MC_GearIn_1(
	Master:= Axis_Spindle  , 
	Slave:=AXIS_1   , 
	Execute:=R_TRIG_5.Q OR ((R_TRIG_1.Q OR R_TRIG_2.Q OR R_TRIG_3.Q) AND HandWheel_3Y) , 
	RatioNumerator:=iMolecule , 
	RatioDenominator:= iDenominator, 
	Acceleration:= 500, 
	Deceleration:= 800, 
	Jerk:= , 
	//BufferMode:= , 
	InGear=> %MX500.5, 
	Busy=> , 
	//Active=> , 
	CommandAborted=> , 
	Error=> , 
	ErrorID=> );
//2轴启动啮合
MC_GearIn_2(
	Master:= Axis_Spindle, 
	Slave:=AXIS_2 , 
	Execute:=R_TRIG_6.Q OR ((R_TRIG_1.Q OR R_TRIG_2.Q OR R_TRIG_3.Q) AND HandWheel_4X) , 
	RatioNumerator:=iMolecule , 
	RatioDenominator:= iDenominator, 
	Acceleration:= 500, 
	Deceleration:= 800, 
	Jerk:= , 
	//BufferMode:= , 
	InGear=> , 
	Busy=> , 
	//Active=> , 
	CommandAborted=> , 
	Error=> , 
	ErrorID=> );
//3轴启动啮合
MC_GearIn_3(
	Master:= Axis_Spindle, 
	Slave:=AXIS_3 , 
	Execute:= R_TRIG_7.Q OR ((R_TRIG_1.Q OR R_TRIG_2.Q OR R_TRIG_3.Q) AND HandWheel_5Z), 
	RatioNumerator:=iMolecule , 
	RatioDenominator:= iDenominator, 
	Acceleration:= 500, 
	Deceleration:= 800, 
	Jerk:= , 
	//BufferMode:= , 
	InGear=> , 
	Busy=> , 
	//Active=> , 
	CommandAborted=> , 
	Error=> , 
	ErrorID=> );
//4轴启动啮合
MC_GearIn_4(
	Master:= Axis_Spindle, 
	Slave:=AXIS_4 , 
	Execute:=  R_TRIG_8.Q OR ((R_TRIG_1.Q OR R_TRIG_2.Q OR R_TRIG_3.Q) AND HandWheel_6X), 
	RatioNumerator:=iMolecule , 
	RatioDenominator:= iDenominator, 
	Acceleration:= 500, 
	Deceleration:= 800, 
	Jerk:= , 
	//BufferMode:= , 
	InGear=> , 
	Busy=> , 
	//Active=> , 
	CommandAborted=> , 
	Error=> , 
	ErrorID=> );
//5轴启动啮合
MC_GearIn_5(
	Master:= Axis_Spindle, 
	Slave:=AXIS_5 , 
	Execute:= R_TRIG_9.Q OR ((R_TRIG_1.Q OR R_TRIG_2.Q OR R_TRIG_3.Q) AND HandWheel_7Y), 
	RatioNumerator:=iMolecule , 
	RatioDenominator:= iDenominator, 
	Acceleration:= 500, 
	Deceleration:= 800, 
	Jerk:= , 
	//BufferMode:= , 
	InGear=> , 
	Busy=> , 
	//Active=> , 
	CommandAborted=> , 
	Error=> , 
	ErrorID=> );
//6轴启动啮合
MC_GearIn_6(
	Master:= Axis_Spindle, 
	Slave:=AXIS_6 , 
	Execute:= R_TRIG_10.Q OR ((R_TRIG_1.Q OR R_TRIG_2.Q OR R_TRIG_3.Q) AND HandWheel_8Y), 
	RatioNumerator:=iMolecule , 
	RatioDenominator:= iDenominator, 
	Acceleration:= 500, 
	Deceleration:= 800, 
	Jerk:= , 
	//BufferMode:= , 
	InGear=> , 
	Busy=> , 
	//Active=> , 
	CommandAborted=> , 
	Error=> , 
	ErrorID=> );
//7轴启动啮合
MC_GearIn_7(
	Master:= Axis_Spindle, 
	Slave:=AXIS_7 , 
	Execute:= R_TRIG_11.Q OR ((R_TRIG_1.Q OR R_TRIG_2.Q OR R_TRIG_3.Q) AND HandWheel_9X), 
	RatioNumerator:=iMolecule , 
	RatioDenominator:= iDenominator, 
	Acceleration:= 500, 
	Deceleration:= 800, 
	Jerk:= , 
	//BufferMode:= , 
	InGear=> , 
	Busy=> , 
	//Active=> , 
	CommandAborted=> , 
	Error=> , 
	ErrorID=> );
//8轴启动啮合
MC_GearIn_8(
	Master:= Axis_Spindle, 
	Slave:=AXIS_8 , 
	Execute:= R_TRIG_12.Q OR ((R_TRIG_1.Q OR R_TRIG_2.Q OR R_TRIG_3.Q) AND HandWheel_10Z), 
	RatioNumerator:=iMolecule , 
	RatioDenominator:= iDenominator, 
	Acceleration:= 500, 
	Deceleration:= 800, 
	Jerk:= , 
	//BufferMode:= , 
	InGear=> , 
	Busy=> , 
	//Active=> , 
	CommandAborted=> , 
	Error=> , 
	ErrorID=> );
//9轴启动啮合
MC_GearIn_9(
	Master:= Axis_Spindle, 
	Slave:=AXIS_9 , 
	Execute:=  R_TRIG_13.Q OR ((R_TRIG_1.Q OR R_TRIG_2.Q OR R_TRIG_3.Q) AND HandWheel_11Y), 
	RatioNumerator:=iMolecule , 
	RatioDenominator:= iDenominator, 
	Acceleration:= 500, 
	Deceleration:= 800, 
	Jerk:= , 
	//BufferMode:= , 
	InGear=> , 
	Busy=> , 
	//Active=> , 
	CommandAborted=> , 
	Error=> , 
	ErrorID=> );

Error :=MC_GearIn_1.Error OR MC_GearIn_2.Error OR MC_GearIn_3.Error OR MC_GearIn_4.Error OR MC_GearIn_5.Error OR MC_GearIn_6.Error OR MC_GearIn_7.Error OR MC_GearIn_8.Error OR MC_GearIn_9.Error ;  
ErrorID :=MC_GearIn_1.ErrorID OR MC_GearIn_2.ErrorID OR MC_GearIn_3.ErrorID OR MC_GearIn_4.ErrorID OR MC_GearIn_5.ErrorID OR MC_GearIn_6.ErrorID OR MC_GearIn_7.ErrorID OR MC_GearIn_8.ErrorID OR MC_GearIn_9.ErrorID ;  

//1轴断开齿合
MC_GearOut_1(Slave:=AXIS_1 , Execute:= F_TRIG_1.Q AND MC_GearIn_1.InGear , Done=> xStop_1 , Busy=> , Error=> , ErrorID=> );

//2轴断开齿合
MC_GearOut_2(Slave:=AXIS_2 , Execute:= F_TRIG_2.Q AND MC_GearIn_2.InGear , Done=> xStop_2 , Busy=> , Error=> , ErrorID=> );

//3轴断开齿合
MC_GearOut_3(Slave:=AXIS_3 , Execute:= F_TRIG_3.Q AND MC_GearIn_3.InGear , Done=> xStop_3 , Busy=> , Error=> , ErrorID=> );


//4轴断开齿合
MC_GearOut_4(Slave:=AXIS_4 , Execute:= F_TRIG_4.Q AND MC_GearIn_4.InGear , Done=> xStop_4 , Busy=> , Error=> , ErrorID=> );


//5轴断开齿合
MC_GearOut_5(Slave:=AXIS_5 , Execute:= F_TRIG_5.Q AND MC_GearIn_5.InGear , Done=> xStop_5 , Busy=> , Error=> , ErrorID=> );


//6轴断开齿合
MC_GearOut_6(Slave:=AXIS_6 , Execute:= F_TRIG_6.Q AND MC_GearIn_6.InGear , Done=> xStop_6 , Busy=> , Error=> , ErrorID=> );


//7轴断开齿合
MC_GearOut_7(Slave:=AXIS_7 , Execute:= F_TRIG_7.Q AND MC_GearIn_7.InGear , Done=> xStop_7 , Busy=> , Error=> , ErrorID=> );


//8断开齿合
MC_GearOut_8(Slave:=AXIS_8 , Execute:= F_TRIG_8.Q AND MC_GearIn_8.InGear , Done=> xStop_8 , Busy=> , Error=> , ErrorID=> );


//9轴断开齿合
MC_GearOut_9(Slave:=AXIS_9 , Execute:= F_TRIG_9.Q AND MC_GearIn_9.InGear , Done=> xStop_9 , Busy=> , Error=> , ErrorID=> );

END_FUNCTION_BLOCK

// Device/Application/30_Ethercat任务/PLC_CNC
PROGRAM PLC_CNC
VAR
	SMC_Interpolator: SMC_Interpolator;
	SMC_ControlAxisByPos1: SMC_ControlAxisByPos;
	SMC_ControlAxisByPos2: SMC_ControlAxisByPos;
	SMC_ControlAxisByPos3: SMC_ControlAxisByPos;
	SMC_TRAFO_Gantry3: SMC_TRAFO_Gantry3;
	SMC_TRAFOF_Gantry3: SMC_TRAFOF_Gantry3;
	SMC_NCDecoder_0: SMC_NCDecoder;
	SMC_CheckVelocities: SMC_CheckVelocities;
	SMC_SmoothPath: SMC_SmoothPath;
	SR: SR;
	RS: RS;
END_VAR
VAR // added by the converter: edge detectors and wires of the graphical bodies
    _w1, _w2, _w3 : BOOL;
    _w4, _w5 : ANY;
END_VAR

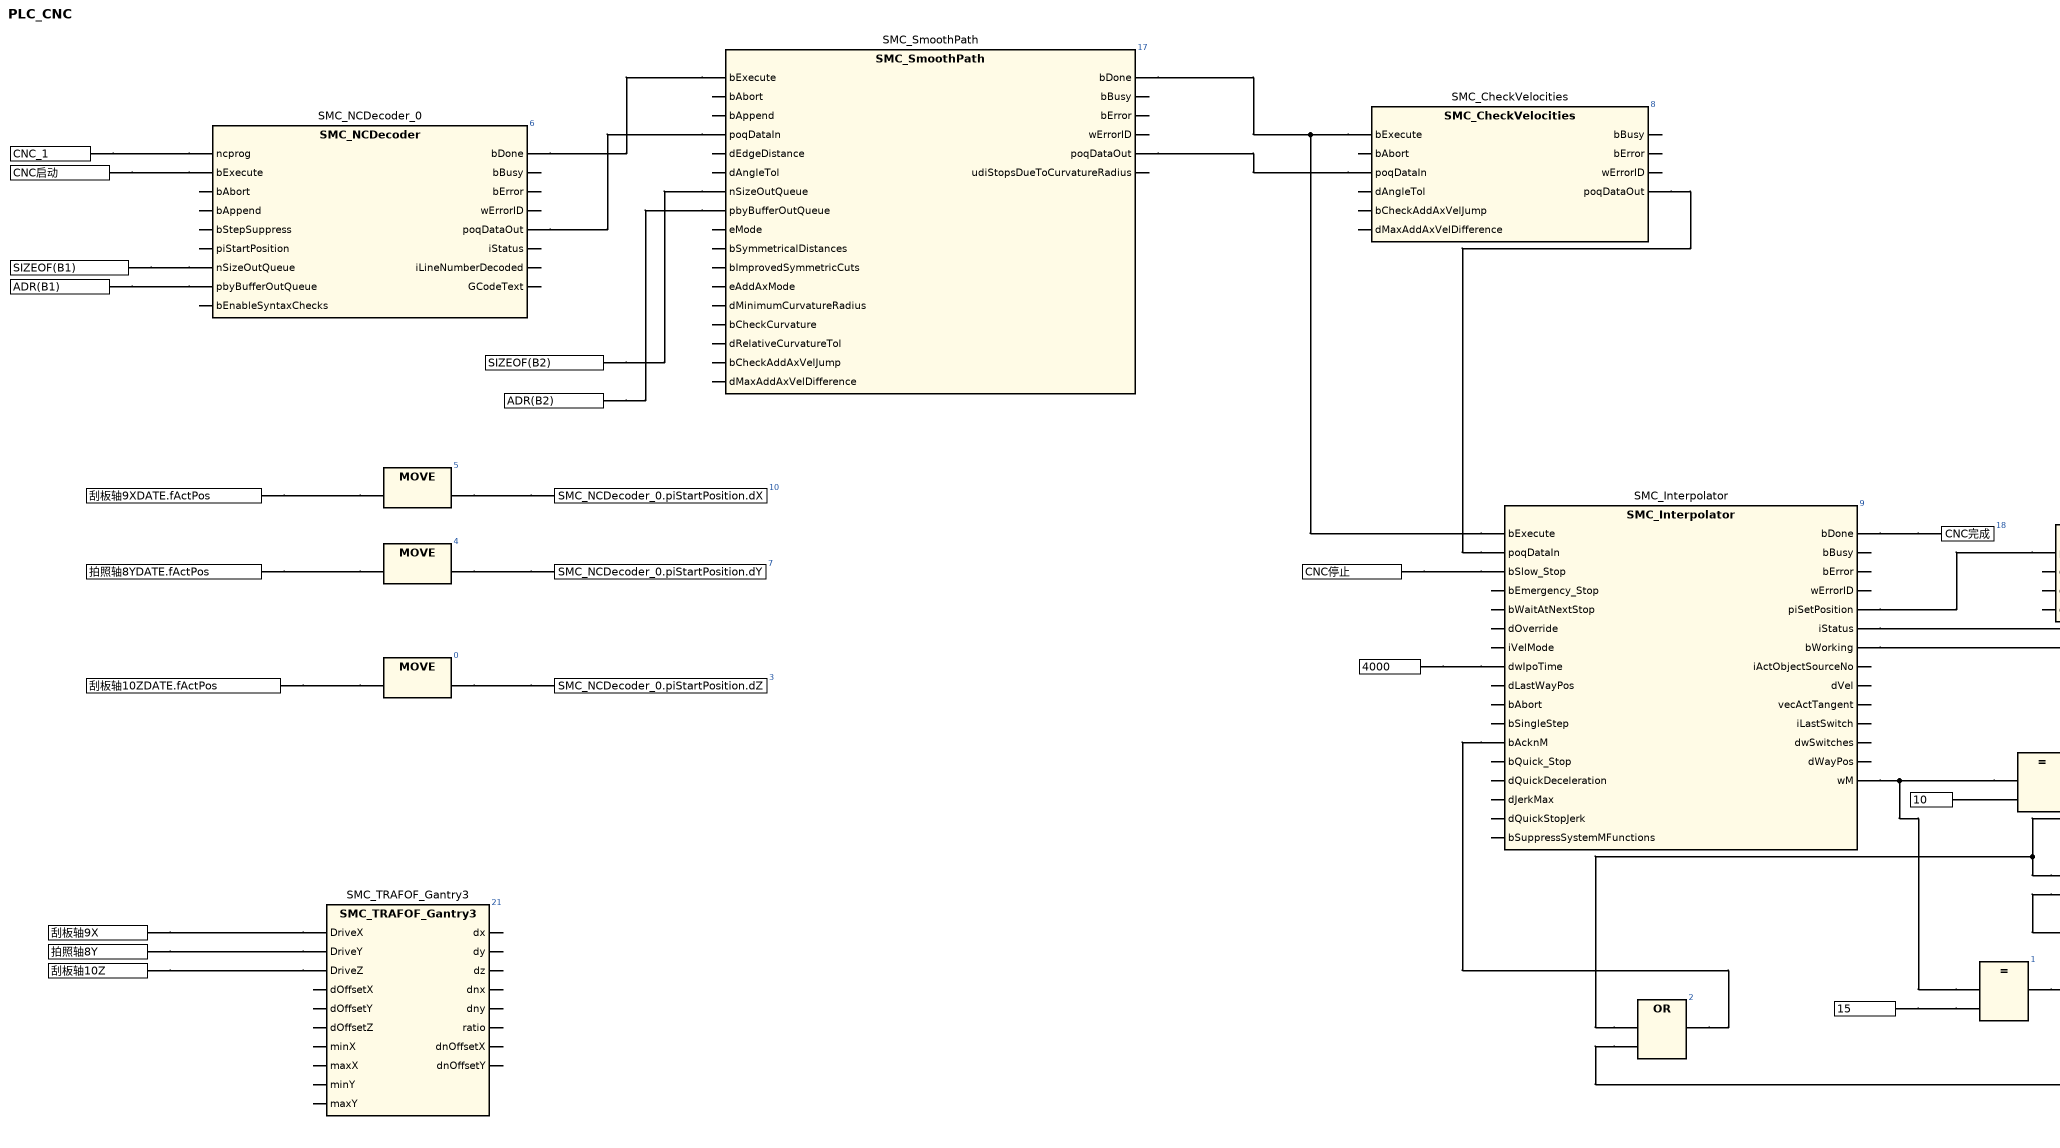
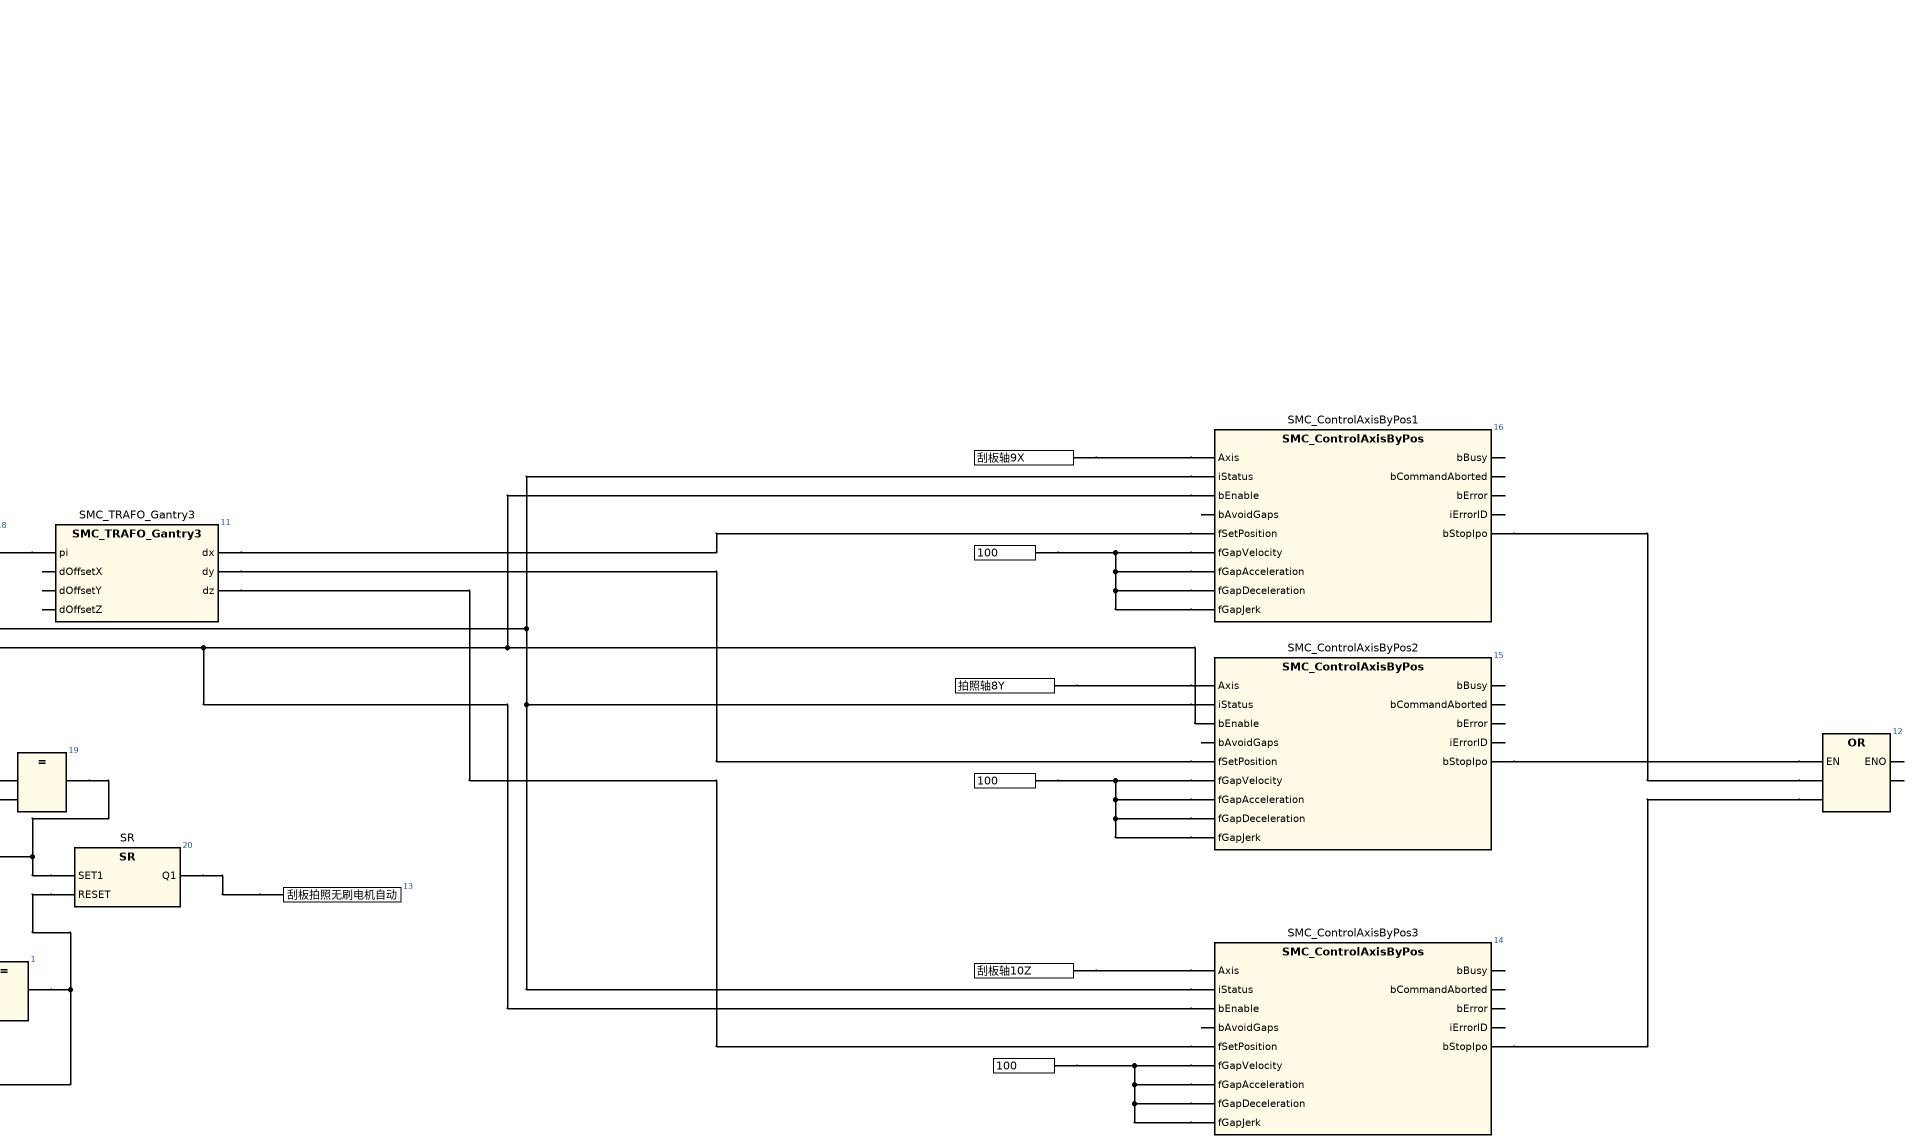
// note: 4 stored wires end on pins the file does not list and are not shown
_w1 := SMC_Interpolator.wM = 15;
_w3 := _w2 OR _w1;
SMC_NCDecoder_0.piStartPosition.dZ := 刮板轴10ZDATE.fActPos;
_w4 := 拍照轴8YDATE.fActPos;
_w5 := 刮板轴9XDATE.fActPos;
SMC_NCDecoder_0(
    ncprog := CNC_1,
    bExecute := CNC启动,
    nSizeOutQueue := SIZEOF(B1),
    pbyBufferOutQueue := ADR(B1)); // SMC_NCDecoder
SMC_NCDecoder_0.piStartPosition.dY := _w4;
SMC_CheckVelocities(bExecute := SMC_SmoothPath.bDone, poqDataIn := SMC_SmoothPath.poqDataOut);
SMC_Interpolator(
    bExecute := SMC_SmoothPath.bDone,
    poqDataIn := SMC_CheckVelocities.poqDataOut,
    bSlow_Stop := CNC停止,
    dwIpoTime := 4000,
    bAcknM := _w3);
SMC_NCDecoder_0.piStartPosition.dX := _w5;
SMC_TRAFO_Gantry3(pi := SMC_Interpolator.piSetPosition);
IF SMC_ControlAxisByPos2.bStopIpo THEN (* SMC_ControlAxisByPos1.bStopIpo OR SMC_ControlAxisByPos3.bStopIpo; result not used *) END_IF
刮板拍照无刷电机自动 := SR.Q1;
SMC_ControlAxisByPos3(
    Axis := 刮板轴10Z,
    iStatus := SMC_Interpolator.iStatus,
    bEnable := SMC_Interpolator.bWorking,
    fSetPosition := SMC_TRAFO_Gantry3.dz,
    fGapVelocity := 100,
    fGapAcceleration := 100,
    fGapDeceleration := 100,
    fGapJerk := 100); // SMC_ControlAxisByPos
SMC_ControlAxisByPos2(
    Axis := 拍照轴8Y,
    iStatus := SMC_Interpolator.iStatus,
    bEnable := SMC_Interpolator.bWorking,
    fSetPosition := SMC_TRAFO_Gantry3.dy,
    fGapVelocity := 100,
    fGapAcceleration := 100,
    fGapDeceleration := 100,
    fGapJerk := 100); // SMC_ControlAxisByPos
SMC_ControlAxisByPos1(
    Axis := 刮板轴9X,
    iStatus := SMC_Interpolator.iStatus,
    bEnable := SMC_Interpolator.bWorking,
    fSetPosition := SMC_TRAFO_Gantry3.dx,
    fGapVelocity := 100,
    fGapAcceleration := 100,
    fGapDeceleration := 100,
    fGapJerk := 100); // SMC_ControlAxisByPos
SMC_SmoothPath(
    bExecute := SMC_NCDecoder_0.bDone,
    poqDataIn := SMC_NCDecoder_0.poqDataOut,
    nSizeOutQueue := SIZEOF(B2),
    pbyBufferOutQueue := ADR(B2));
CNC完成 := SMC_Interpolator.bDone;
_w2 := SMC_Interpolator.wM = 10;
SR(SET1 := _w2, RESET := _w1);
SMC_TRAFOF_Gantry3(DriveX := 刮板轴9X, DriveY := 拍照轴8Y, DriveZ := 刮板轴10Z);

END_PROGRAM

// Device/Application/40_Man/PLC_MainPRG
PROGRAM PLC_MainPRG

VAR
	PLC_Mode_0: FB_Mode;
	TON_1: TON;
	RB_Control_0: FB_RB_Control;
	TON_0: TON;
	TON_2: TON;
	TON_3: TON;
	SysHC_ModbusTcpSlaveDiagnose_0: SysHC_ModbusTcpSlaveDiagnose;
	点样step: INT;
	打样伺服移动step: INT;
END_VAR

IF 点样测试 THEN
	CASE 打样伺服移动step OF
		
		0:
			点样轴6XDATE.fAbsTarget:=HMI_点样轴6X.position[2];        //起始位
			点样轴6XDATE.xMoveAbs:=TRUE;
			打样伺服移动step:=20;
		20:
			IF 点样轴6XDATE.bAbMoveDone THEN
				
				打样伺服移动step:=30;
				点样轴6XDATE.xMoveAbs:=FALSE;
			END_IF
		30:
			点样轴6XDATE.fAbsTarget:=HMI_点样轴6X.position[3];             //终点位
			点样轴6XDATE.xMoveAbs:=TRUE;
			打样伺服移动step:=40;
		40:
			IF 点样轴6XDATE.bAbMoveDone THEN
				
				打样伺服移动step:=0;
				点样轴6XDATE.xMoveAbs:=FALSE;
			END_IF
			
	END_CASE
ELSE
	打样伺服移动step:=0;
END_IF







A00_设备状态显示及控制 ();

A20_机器人();
%MW1000:=0;

PLC_Cyinder_气缸动作();

CASE MODE_State OF
	EN_功能块状态.运行:
		A10_上下料伺服流程 ();
		Sample_point_sampling_上样点样();
		Collection_process_收集流程();
		Expand_process_展开流程();
		Photo_scraper_拍照刮板();
		Robotic_Process_机器人流程();
		Develop_TankDrain();
	IF NOT 上料进料传感器 THEN
		Alarm.2:=TRUE;
	END_IF
	IF NOT 下料出料传感器 THEN
		Alarm.3:=TRUE;
	END_IF
END_CASE




//所有状态复位
TON_3(IN:=复位,PT:=T#5S );
IF NOT 急停 OR TON_3.Q THEN
	A30_急停();
END_IF





//升降伺服流程
IF MODE_State<>1 THEN
	伺服上料_Setp:=0;
	伺服下料_Setp:=0;
END_IF






//检测MODBUS通讯
SysHC_ModbusTcpSlaveDiagnose_0(
	xEnable:=TRUE , 
	strSlaveIP:= '192.168.0.15', 
	xValid=> , 
	xBusy=> , 
	xError=> , 
	eErrorID=> , 
	stDiagData=>ModbusTcpError );

ACTION A30_急停:

伺服上料_Setp:=0;
伺服下料_Setp:=0;
//收集工位
收集下压气缸手动:=FALSE;
收集下压气缸自动:=FALSE;
收集夹持气缸手动:=FALSE;
收集夹持气缸自动:=FALSE;
收集升降气缸手动:=FALSE;
收集升降气缸自动:=FALSE;
收集伸缩气缸手动:=FALSE;
收集伸缩气缸自动:=FALSE;
收集进液手动:=FALSE;
收集进液自动:=FALSE;
收集排液手动:=FALSE;
收集排液自动:=FALSE;
收集正压排液手动:=FALSE;
收集正压排液自动:=FALSE;
溶液收集瓶定位手动:=FALSE;
收集工位允许放收集瓶:=FALSE;
收集工位允许放收集器:=FALSE;
收集工位允许机器人退出工位:=FALSE;
收集工位允许机器人取收集瓶放暂存工位:=FALSE;
收集工位允许取收集器:=FALSE;
收集工位机器人取收集器放回暂存工位:=FALSE;
collect_prepare_OK:=FALSE;
collect_OK:=FALSE;
收集工位放收集器完成:=FALSE;
收集工位放收集瓶完成:=FALSE;
收集工位放收集器到工位:=FALSE;

收集工位机器人退出完成:=FALSE;

收集工位机器人放收集瓶到暂存工位完成:=FALSE;

收集工位机器人到达收集器位置:=FALSE;
//展开工位
expand_initialization_OK:=FALSE;
Expand_Group_clean_OK:=FALSE;
Expand_up_liquid_OK:=FALSE;
Expand_silica_gel_plate_OK:=FALSE;
展开工位允许放硅胶板:=FALSE;
展开工位允许取硅胶板:=FALSE;
展开工位机器人到达准备点:=FALSE;
展开工位机器人放硅胶板完成:=FALSE;
展开工位取硅胶板完成:=FALSE;
展开工位允许放硅胶板1:=FALSE;
展缸1气缸1手动:=FALSE;
展缸1气缸1自动:=FALSE;
展缸1进液电池阀1手动:=FALSE;
展缸1进液电池阀1自动:=FALSE;
展缸1排液电池阀1手动:=FALSE;
展缸1排液电池阀1自动:=FALSE;
展缸1吹气电池阀1手动:=FALSE;
展缸1吹气电池阀1自动:=FALSE;
展缸1气缸2手动:=FALSE;
展缸1气缸2自动:=FALSE;
展缸1进液电池阀2手动:=FALSE;
展缸1进液电池阀2自动:=FALSE;
展缸1排液电池阀2手动:=FALSE;
展缸1排液电池阀2自动:=FALSE;
展缸1吹气电池阀2手动:=FALSE;
展缸1吹气电池阀2自动:=FALSE;
展缸1气缸3手动:=FALSE;
展缸1气缸3自动:=FALSE;
展缸1进液电池阀3手动:=FALSE;
展缸1进液电池阀3自动:=FALSE;	
展缸1排液电池阀3手动:=FALSE;
展缸1排液电池阀3自动:=FALSE;
展缸1吹气电池阀3手动:=FALSE;
展缸1吹气电池阀3自动:=FALSE;
展缸1气缸4手动:=FALSE;
展缸1气缸4自动:=FALSE;
展缸1进液电池阀4手动:=FALSE;
展缸1进液电池阀4自动:=FALSE;	
展缸1排液电池阀4手动:=FALSE;
展缸1排液电池阀4自动:=FALSE;
展缸1吹气电池阀4手动:=FALSE;
展缸1吹气电池阀4自动:=FALSE;
展缸2气缸1手动:=FALSE;
展缸2气缸1自动:=FALSE;
展缸2进液电池阀1手动:=FALSE;
展缸2进液电池阀1自动:=FALSE;
展缸2排液电池阀1手动:=FALSE;
展缸2排液电池阀1自动:=FALSE;
展缸2吹气电池阀1手动:=FALSE;
展缸2吹气电池阀1自动:=FALSE;
展缸2气缸2手动:=FALSE;
展缸2气缸2自动:=FALSE;
展缸2进液电池阀2手动:=FALSE;
展缸2进液电池阀2自动:=FALSE;
展缸2排液电池阀2手动:=FALSE;
展缸2排液电池阀2自动:=FALSE;
展缸2吹气电池阀2手动:=FALSE;
展缸2吹气电池阀2自动:=FALSE;
展缸2气缸3手动:=FALSE;
展缸2气缸3自动:=FALSE;
展缸2进液电池阀3手动:=FALSE;
展缸2进液电池阀3自动:=FALSE;	
展缸2排液电池阀3手动:=FALSE;
展缸2排液电池阀3自动:=FALSE;
展缸2吹气电池阀3手动:=FALSE;
展缸2吹气电池阀3自动:=FALSE;
展缸2气缸4手动:=FALSE;
展缸2气缸4自动:=FALSE;
展缸2进液电池阀4手动:=FALSE;
展缸2进液电池阀4自动:=FALSE;	
展缸2排液电池阀4手动:=FALSE;
展缸2排液电池阀4自动:=FALSE;
展缸2吹气电池阀4手动:=FALSE;
展缸2吹气电池阀4自动:=FALSE;
Expand_Step:=0;
//拍照刮板
刮板拍照真空自动:=FALSE;
刮板拍照真空手动:=FALSE;
刮板拍照无刷电机手动:=FALSE;
刮板拍照无刷电机自动:=FALSE;
刮板拍照定位气缸手动:=FALSE;
刮板拍照定位气缸自动:=FALSE;
粉末收集器定位手动:=FALSE;
粉末收集器定位自动:=FALSE;
刮板拍照遮光气缸手动:=FALSE;
刮板拍照遮光气缸自动:=FALSE;
刮板拍照旋转气缸手动:=FALSE;
刮板拍照旋转气缸自动:=FALSE;
刮板拍照下压气缸手动:=FALSE;
刮板拍照下压气缸自动:=FALSE;
拍照工位允许放硅胶板:=FALSE;
拍照工位允许放收集器:=FALSE;
拍照工位机器人退出工位:=FALSE;
拍照工位允许取收集器:=FALSE;
拍照工位机器人退出:=FALSE;
拍照工位放硅胶板完成 := FALSE;
 scrape_IsLast := FALSE;       // ★ 新增		
拍照工位机器人到达夹持位 := FALSE;
scrape_PhotoMode:=0;
拍照工位机器人退出工位完成 := FALSE;
刮板拍照工位站位符:=FALSE;
拍照工位机器人到达收集器夹持位 := FALSE;
scrape_Step:=0;
拍照工位机器人退出完成 := FALSE;
拍照工位允许取硅胶板放废料区 := FALSE;
拍照工位允许取硅胶板去展开 := FALSE;
拍照工位机器人取硅胶板完成 := FALSE;
scrape_WaitConfirm := FALSE;
Camera_scraper_initialization_OK:=FALSE;
Photo_preparation_completed_OK:=FALSE;
Scraper_collection_completed:=FALSE;
Robot_completes_material_retrieval:=FALSE;	
取拍照硅胶完step:=0;

//上样点样
上样定位手动:=FALSE;
上样定位自动:=FALSE;
上样点样三通电池阀手动:=FALSE;
上样点样三通电池阀自动:=FALSE;
上样吹气手动:=FALSE;
上样吹气自动:=FALSE;
打样瓶上料轴3YDATE.fAbsTarget:=0;
点样轴6XDATE.fAbsTarget:=0;
点样轴7YDATE.fAbsTarget:=0;
上样轴4X轴DATE.fAbsTarget:=0;
上样轴5Z轴DATE.fAbsTarget:=0;
上样点样允许放硅胶板:=FALSE;
点样轴7YDATE.xMoveAbs:=FALSE;
点样轴6XDATE.xMoveAbs:=FALSE;
上样轴5Z轴DATE.xMoveAbs:=FALSE;
上样轴4X轴DATE.xMoveAbs:=FALSE;
打样瓶上料轴3YDATE.xMoveAbs:=FALSE;
Sampling_Spray_sample_OK:=FALSE;
Sampling_liquid_absorption:=FALSE;
Sampling_preparation_OK:=FALSE;
上样点样允许取硅胶板:=FALSE;
上样点样放硅胶板完成:=FALSE;
大真空泵站位[11]:=FALSE;
大真空泵自动:=FALSE;
Sampling_Step:=0;

//机器人
Execute:=0;
FunctionID:=0;
ParameterList1:=0;
ParameterList2:=0;
ParameterList3:=0;
ParameterList4:=0;
ParameterList5:=0;
ParameterList6:=0;
ParameterList7:=0;
ParameterList8:=0;
ParameterList9:=0;
ParameterList10:=0;

RO_ParameterList1:=0;
RO_ParameterList2:=0;
RO_ParameterList4:=0;
RO_ParameterList5:=0;
RO_ParameterList6:=0;
RO_ParameterList7:=0;
RO_ParameterList8:=0;
RO_ParameterList9:=0;
RO_ParameterList10:=0;
升降上料机器人取料完成:=FALSE;
泵站位符:=FALSE;
上样料架报警:=FALSE;
取工具setp:=0;
取工具完成:=FALSE;
取升降硅胶板step:=0;
取升降硅胶板完成:=FALSE;
放点样硅胶板step:=0;
放点样硅胶板完成:=FALSE;
取点样硅胶板step:=0;
取点样硅胶板完成:=FALSE;
放展缸硅胶板完成:=FALSE;
放展缸硅胶板step:=0;
取展缸硅胶板step:=0;
取展缸硅胶板完成:=FALSE;
放拍照硅胶板完成:=FALSE;
放拍照硅胶板step:=0;
取收集器组放暂存工位step:=0;
取收集瓶组放暂存工位完成:=FALSE;
取暂存收集器放刮板位完成:=FALSE;
取暂存收集器放刮板位step:=0;
取刮板收集器放到收集工位完成:=FALSE;
取刮板收集器放到收集工位step:=0;
取暂存收集瓶放收集工位step:=0;
取暂存收集瓶放收集工位完成:=FALSE;
取收集器放暂存工位完成:=FALSE;
取收集器放暂存工位step:=0;
取刮板硅胶板放废料区step:=0;
取刮板硅胶板放废料区完成:=FALSE;
取暂存收集器组放仓库完成:=FALSE;
取暂存收集器组放仓库step:=0;
取收集器组放暂存工位完成:=FALSE;
取收集瓶组放暂存工位step:=0;
取暂存收集瓶组放仓库完成:=FALSE;
取暂存收集瓶组放仓库step:=0;
取收集瓶放暂存工位step:=0;
取收集瓶放暂存工位完成:=FALSE;
机器人流程:=0;
溶液收集瓶定位自动:=FALSE;
溶液收集瓶定位手动:=FALSE;
END_ACTION

ACTION A20_机器人:
//机器人远程控制
RB_Control_0(
    PowerOn := RB_使能状态, 
    PowerOnOut =>RB_上使能 , 

    ResetOut =>RB_复位 , 

    Reset := 复位, 

    StartCmd := 启动, 
    StopCmd :=  TON_3.Q OR NOT 急停, 
    PauseCmd := NOT 停止, 
    RobotRunning := RB_运行中, 
    RobotStopped :=RB_停止中 , 
    RobotPaused :=RB_暂停中 , 
    RobotAlarm :=RB_报警中 , 
    StartOut =>RB_启动 , 
    StopOut => RB_停止, 
    PauseOut =>  RB_暂停, 
    StatusRun => , 
    StatusStop => , 
    StatusPause => , 
    StatusAlarm => , 

	);
END_ACTION

ACTION A00_设备状态显示及控制:
//PLC模式切换
PLC_Mode_0(
    bWarning_alarm := cyinderAlarm<>0 OR Alarm<>0 OR 上样料架报警 OR ModbusTcpError.byDiagData>0, 

	xStart:= 启动 OR PLCStart, 
	xStop:=NOT  停止 OR PLCStop, 
	xReset:=复位  , 
	xAutoMode:=手自动  , 
	xFault:=伺服报警 OR ECAT掉站报警 OR 伺服未回原点报警, 
	xEmergency:= 急停 , 
	bRed=>三色灯红  , 
	bYellow=> 三色灯黄, 
	bGreen=> 三色灯绿, 
	bBuzzer=> 蜂鸣器 , 
	iState=>MODE_STATE  , 
	bAuto=>ManualAuto  );
	
	//伺服报错
IF   玻璃上料轴1ZDATE.bError OR 玻璃上料轴2ZDATE.bError OR 打样瓶上料轴3YDATE.bError OR 点样轴6XDATE.bError OR 点样轴7YDATE.bError OR 拍照轴8YDATE.bError OR 刮板轴9XDATE.bError OR 刮板轴10ZDATE.bError OR 地轨轴11YDATE.bError OR 上样轴4X轴DATE.bError OR 上样轴5Z轴DATE.bError THEN
	伺服报警:=TRUE;
END_IF
   //伺服报错复位
IF 复位 THEN
	伺服报警:=FALSE;
	伺服未回原点报警:=FALSE;
	Alarm:=0;
	cyinderAlarm:=0;
	上样料架报警:=FALSE;
END_IF


IF NOT 玻璃上料轴1ZDATE.bHomed OR NOT 玻璃上料轴2ZDATE.bHomed OR NOT 打样瓶上料轴3YDATE.bHomed OR NOT 点样轴6XDATE.bHomed OR NOT 点样轴7YDATE.bHomed OR NOT 拍照轴8YDATE.bHomed OR NOT 刮板轴9XDATE.bHomed OR NOT 刮板轴10ZDATE.bHomed  OR NOT 地轨轴11YDATE.bHomed OR NOT 上样轴4X轴DATE.bHomed OR NOT 上样轴5Z轴DATE.bHomed THEN
	伺服未回原点报警:=TRUE ;
END_IF
END_ACTION

ACTION A10_上下料伺服流程:
//初始化
IF MODE_State =4 OR  初始化  THEN

		玻璃上料轴1ZDATE.fAbsTarget :=0;
		玻璃上料轴1ZDATE.xMoveAbs:=TRUE;
		玻璃上料轴1ZDATE.xJogPos :=FALSE;
		升降上料伺服允许取料 :=FALSE ;
		升降上料伺服下降完成 :=FALSE ;
		伺服上料_Setp:=0;
		伺服上料_Setp:=0;
		升降下料伺服允许放料  :=FALSE ;
		玻璃上料轴2ZDATE.xJogNeg :=FALSE;
		玻璃上料轴2ZDATE.xJogPos :=FALSE;
		升降上料机器人取料完成:=FALSE;
END_IF



//上料流程
IF MODE_State =1 THEN     //自动模式下
	IF 玻璃上料轴1ZDATE.bHomed AND 玻璃升降接近开关1 AND 上料进料传感器 AND 伺服上料_Setp=0 AND NOT Alarm.0 AND 升降上料完成 THEN
		伺服上料_Setp :=1;
	END_IF
	
    CASE 伺服上料_Setp OF
    	1 :
			IF NOT 玻璃升降光电开关1 AND 玻璃上料轴1ZDATE.fActPos<514  THEN
				Z1JOG_pos :=TRUE;
				ELSE
				Z1JOG_pos :=FALSE;
				伺服上料_Setp:=10;
			END_IF
   
	   10:
		   IF 玻璃升降光电开关1 THEN
		   	升降上料伺服允许取料 :=TRUE;
			伺服上料_Setp:=20;
		   END_IF
		   
	   20:
		   IF 升降上料机器人已吸住物料 THEN
		   	玻璃上料轴1ZDATE.fRelTarget :=-5.0;
			玻璃上料轴1ZDATE.xMoveRel :=TRUE;
			升降上料机器人已吸住物料:=FALSE;
			伺服上料_Setp:=30;
		   END_IF
	   30:
		   IF 玻璃上料轴1ZDATE .bReMoveDone  THEN
		   	升降上料伺服下降完成 :=TRUE ;
			玻璃上料轴1ZDATE.xMoveRel :=FALSE;
			伺服上料_Setp:=40;
		   END_IF
	   40:
		   IF 升降上料机器人取料完成  THEN
		   	升降上料伺服下降完成 :=FALSE ;
			升降上料伺服允许取料 :=FALSE ;
			升降上料机器人取料完成:=FALSE;
			伺服上料_Setp:=1;
		   END_IF 
    END_CASE
	
	IF 玻璃上料轴1ZDATE.fActPos>=510.0 AND  玻璃升降光电开关1 AND  NOT 玻璃升降接近开关1 THEN
		Alarm.0:=TRUE;                                             //上料机构无物料
		升降上料完成:=FALSE;
		玻璃上料轴1ZDATE.fAbsTarget :=0;
		玻璃上料轴1ZDATE.xMoveAbs:=TRUE;
		Z1JOG_pos :=FALSE;
		升降上料伺服允许取料 :=FALSE ;
		升降上料伺服下降完成 :=FALSE ;
		伺服上料_Setp:=0;
	END_IF
	IF 玻璃上料轴1ZDATE .bAbMoveDone  THEN
		玻璃上料轴1ZDATE.xMoveAbs:=FALSE;
		升降上料机器人放料完成:=FALSE;
    END_IF
	
	
END_IF
//下料流程
IF MODE_State =1 THEN     //自动模式下
	IF 玻璃上料轴2ZDATE.bHomed  AND 下料出料传感器 AND 伺服下料_Setp=0 AND NOT Alarm.1 AND 升降下料完成 THEN
		伺服下料_Setp :=1;
	END_IF
	
    CASE 伺服下料_Setp  OF
    	1 :
			IF NOT 玻璃升降光电开关2 AND 玻璃上料轴2ZDATE.fActPos<510  THEN
				Z2JOG_POS :=TRUE;
				
				ELSE
				Z2JOG_POS :=FALSE;
				伺服下料_Setp:=10;
			END_IF
   
	   10:
		   IF 玻璃升降光电开关2 THEN
			   Z2JOG_NEG :=TRUE;
			   伺服下料_Setp:=15;
		   END_IF
	   15:
		   IF NOT 玻璃升降光电开关2  THEN
				升降下料伺服允许放料  :=TRUE;
				Z2JOG_NEG :=FALSE;
				伺服下料_Setp:=20;
		   END_IF
			  
	   
	   20:
		   IF 升降下料机器人放废料完成 AND 玻璃升降光电开关2 AND 玻璃升降接近开关2 THEN
		   	Z2JOG_NEG :=TRUE;
			升降下料伺服允许放料  :=FALSE ;
			升降下料机器人放废料完成:=FALSE;
			伺服下料_Setp:=30;
		   END_IF
		  
	   30:
		   IF NOT 玻璃升降光电开关2 THEN
		   	Z2JOG_NEG :=FALSE;
			取刮板硅胶板放废料区完成:=FALSE;
			伺服下料_Setp:=15;
		   END_IF
	  
    END_CASE
	
	IF 玻璃上料轴2ZDATE.fActPos<=0 AND 玻璃升降光电开关1 THEN
		Alarm.1:=TRUE;                                           //下料机构已满料
		升降下料完成:=FALSE;
		伺服下料_Setp:=0;
		升降下料伺服允许放料  :=FALSE ;
		Z2JOG_NEG :=FALSE;
		Z2JOG_POS :=FALSE;
		玻璃上料轴2ZDATE.fAbsTarget :=0;
		玻璃上料轴2ZDATE.xMoveAbs:=TRUE;
		伺服下料_Setp:=0;
	END_IF
	IF 玻璃上料轴2ZDATE .bAbMoveDone  THEN
		玻璃上料轴2ZDATE.xMoveAbs:=FALSE;
		升降下料伺服允许放料  :=FALSE ;
    END_IF
END_IF
END_ACTION

END_PROGRAM

// Device/Application/40_Man/PLC_Cyinder_气缸动作
PROGRAM PLC_Cyinder_气缸动作
VAR
	cylinder_0: FB_cylinder;
	cylinder_1: FB_cylinder;
	cylinder_2: FB_cylinder;
	cylinder_3 :FB_cylinder ;
	cylinder_4 :FB_cylinder ;
	cylinder_5 :FB_cylinder ;
	cylinder_6 :FB_cylinder ;
	cylinder_7 :FB_cylinder ;
	cylinder_8 :FB_cylinder ;
	cylinder_9 :FB_cylinder ;
	cylinder_10 :FB_cylinder ;
	cylinder_11 :FB_cylinder ;
	cylinder_12 :FB_cylinder ;
	cylinder_13 :FB_cylinder ;
	cylinder_14 :FB_cylinder ;
	cylinder_15 :FB_cylinder ;
	cylinder_16 :FB_cylinder ;
	cylinder_17 :FB_cylinder ;
	cylinder_18 :FB_cylinder ;
	cylinder_19 :FB_cylinder ;
	cylinder_20 :FB_cylinder ;
	cylinder_21 :FB_cylinder ;
	cylinder_22 :FB_cylinder ;
	cylinder_23 :FB_cylinder ;
	cylinder_24 :FB_cylinder ;
	cylinder_25 :FB_cylinder ;
	cylinder_26 :FB_cylinder ;
	cylinder_27 :FB_cylinder ;
	cylinder_28 :FB_cylinder ;
	cylinder_29 :FB_cylinder ;
	cylinder_30 :FB_cylinder ;
	cylinder_31 :FB_cylinder ;
	cylinder_32 :FB_cylinder ;
	cylinder_33 :FB_cylinder ;
	cylinder_34 :FB_cylinder ;
	cylinder_35 :FB_cylinder ;
	cylinder_36 :FB_cylinder ;
	cylinder_37 :FB_cylinder ;
	cylinder_38 :FB_cylinder ;
	cylinder_39 :FB_cylinder ;
	cylinder_40 :FB_cylinder ;
	cylinder_41 :FB_cylinder ;
	cylinder_42 :FB_cylinder ;
	cylinder_43 :FB_cylinder ;
	cylinder_44 :FB_cylinder ;
	cylinder_45 :FB_cylinder ;
	cylinder_46 :FB_cylinder ;
	cylinder_47 :FB_cylinder ;
	cylinder_48 :FB_cylinder ;
	cylinder_49 :FB_cylinder ;
	cylinder_50 :FB_cylinder ;
END_VAR

//气缸动作
//展缸1气缸1
cylinder_0(
    xManualRetract := , 
    xAutoRetract := , 
    yValve2 => , 
    cylinder_type := 0, 

	xManualAuto:=ManualAuto  , 
	xManualExtend:=展缸1气缸1手动 , 
	xAutoExtend:= 展缸1气缸1自动, 
	xReset:=复位  , 
	xPosExtend:= 展缸1气缸1原点, 
	xPosRetract:= 展缸1气缸1动点 , 
	tTimeout:= T#5S, 
	yValve1=> 展缸1气缸1 , 
	bAlarm=> cyinderAlarm.0);
//展缸1气缸2
cylinder_1(
    xManualRetract := , 
    xAutoRetract := , 
    yValve2 => , 
    cylinder_type :=0 , 

	xManualAuto:=ManualAuto  , 
	xManualExtend:=展缸1气缸2手动 , 
	xAutoExtend:= 展缸1气缸2自动, 
	xReset:=复位  , 
	xPosExtend:= 展缸1气缸2原点, 
	xPosRetract:= 展缸1气缸2动点 , 
	tTimeout:= T#5S, 
	yValve1=> 展缸1气缸2, 
	bAlarm=> cyinderAlarm.1);
//展缸1气缸3
cylinder_2(
    xManualRetract := , 
    xAutoRetract := , 
    yValve2 => , 
    cylinder_type := 0, 

	xManualAuto:=ManualAuto  , 
	xManualExtend:=展缸1气缸3手动 , 
	xAutoExtend:= 展缸1气缸3自动, 
	xReset:=复位  , 
	xPosExtend:= 展缸1气缸3原点, 
	xPosRetract:= 展缸1气缸3动点 , 
	tTimeout:= T#5S, 
	yValve1=> 展缸1气缸3, 
	bAlarm=> cyinderAlarm.2);
//展缸1气缸4
cylinder_3(
    xManualRetract := , 
    xAutoRetract := , 
    yValve2 => , 
    cylinder_type :=0 , 

	xManualAuto:=ManualAuto  , 
	xManualExtend:=展缸1气缸4手动 , 
	xAutoExtend:= 展缸1气缸4自动, 
	xReset:=复位  , 
	xPosExtend:= 展缸1气缸4原点, 
	xPosRetract:= 展缸1气缸4动点 , 
	tTimeout:= T#5S, 
	yValve1=> 展缸1气缸4, 
	bAlarm=> cyinderAlarm.3);
//展缸2气缸1
cylinder_4(
    xManualRetract := , 
    xAutoRetract := , 
    yValve2 => , 
    cylinder_type := 0, 

	xManualAuto:=ManualAuto  , 
	xManualExtend:=展缸2气缸1手动 , 
	xAutoExtend:= 展缸2气缸1自动, 
	xReset:=复位  , 
	xPosExtend:= 展缸2气缸1原点, 
	xPosRetract:= 展缸2气缸1动点 , 
	tTimeout:= T#5S, 
	yValve1=> 展缸2气缸1, 
	bAlarm=> cyinderAlarm.4);
//展缸2气缸2
cylinder_5(
    xManualRetract := , 
    xAutoRetract := , 
    yValve2 => , 
    cylinder_type :=0 , 

	xManualAuto:=ManualAuto  , 
	xManualExtend:=展缸2气缸2手动 , 
	xAutoExtend:= 展缸2气缸2自动, 
	xReset:=复位  , 
	xPosExtend:= 展缸2气缸2原点, 
	xPosRetract:= 展缸2气缸2动点 , 
	tTimeout:= T#5S, 
	yValve1=> 展缸2气缸2, 
	bAlarm=> cyinderAlarm.5);
//展缸2气缸3
cylinder_6(
    xManualRetract := , 
    xAutoRetract := , 
    yValve2 => , 
    cylinder_type := 0, 

	xManualAuto:=ManualAuto  , 
	xManualExtend:=展缸2气缸3手动 , 
	xAutoExtend:= 展缸2气缸3自动, 
	xReset:=复位  , 
	xPosExtend:= 展缸2气缸3原点, 
	xPosRetract:= 展缸2气缸3动点 , 
	tTimeout:= T#5S, 
	yValve1=> 展缸2气缸3, 
	bAlarm=> cyinderAlarm.6);
//展缸2气缸4
cylinder_7(
    xManualRetract := , 
    xAutoRetract := , 
    yValve2 => , 
    cylinder_type := 0, 

	xManualAuto:=ManualAuto  , 
	xManualExtend:=展缸2气缸4手动 , 
	xAutoExtend:= 展缸2气缸4自动, 
	xReset:=复位  , 
	xPosExtend:= 展缸2气缸4原点, 
	xPosRetract:= 展缸2气缸4动点 , 
	tTimeout:= T#5S, 
	yValve1=> 展缸2气缸4, 
	bAlarm=> cyinderAlarm.7);
//大真空泵
cylinder_8(
    xManualRetract := , 
    xAutoRetract := , 
    yValve2 => , 
    cylinder_type :=0 , 

	xManualAuto:=ManualAuto  , 
	xManualExtend:= 大真空泵手动, 
	xAutoExtend:= 大真空泵自动, 
	xReset:=复位  , 
	xPosExtend:= , 
	xPosRetract:=  , 
	tTimeout:= , 
	yValve1=> 大真空泵, 
	bAlarm=> );
//收集平台下压气缸
cylinder_9(
    xManualRetract := , 
    xAutoRetract := , 
    yValve2 => , 
    cylinder_type := 0, 

	xManualAuto:=ManualAuto  , 
	xManualExtend:= 收集下压气缸手动, 
	xAutoExtend:= 收集下压气缸自动, 
	xReset:=复位  , 
	xPosExtend:=收集平台下压气缸原点 , 
	xPosRetract:= 收集下压气缸手动 OR 收集下压气缸自动, 
	tTimeout:= T#5S, 
	yValve1=> 收集下压气缸 , 
	bAlarm=> cyinderAlarm.8);
//收集平台夹持气缸
cylinder_10(
    xManualRetract := , 
    xAutoRetract := , 
    yValve2 => , 
    cylinder_type := 0, 

	xManualAuto:=ManualAuto  , 
	xManualExtend:= 收集夹持气缸手动, 
	xAutoExtend:= 收集夹持气缸自动, 
	xReset:=复位  , 
	xPosExtend:=收集平台夹持气缸原点 , 
	xPosRetract:= 收集平台夹持气缸动点, 
	tTimeout:= T#5S, 
	yValve1=> 收集夹持气缸  , 
	bAlarm=> cyinderAlarm.9);	
//收集平台升降气缸
cylinder_11(
    xManualRetract := , 
    xAutoRetract := , 
    yValve2 => , 
    cylinder_type := 0, 

	xManualAuto:=ManualAuto  , 
	xManualExtend:= 收集升降气缸手动, 
	xAutoExtend:= 收集升降气缸自动, 
	xReset:=复位  , 
	xPosExtend:=收集平台升降气缸原点 , 
	xPosRetract:= 收集平台升降气缸动点, 
	tTimeout:= T#5S, 
	yValve1=> 收集升降气缸   , 
	bAlarm=> cyinderAlarm.10);	
//收集平台伸缩气缸
cylinder_12(
    xManualRetract := , 
    xAutoRetract := , 
    yValve2 => , 
    cylinder_type :=0 , 

	xManualAuto:=ManualAuto  , 
	xManualExtend:= 收集伸缩气缸手动, 
	xAutoExtend:= 收集伸缩气缸自动, 
	xReset:=复位, 
	xPosExtend:=收集平台推出气缸原点, 
	xPosRetract:= 收集平台推出气缸动点, 
	tTimeout:= T#5S, 
	yValve1=> 收集伸缩气缸, 
	bAlarm=> cyinderAlarm.11);		
//刮板拍照遮光气缸
cylinder_13(
    xManualRetract := , 
    xAutoRetract := , 
    yValve2 => , 
    cylinder_type :=0 , 

	xManualAuto:=ManualAuto  , 
	xManualExtend:= 刮板拍照遮光气缸手动, 
	xAutoExtend:=刮板拍照遮光气缸自动 , 
	xReset:=复位  , 
	xPosExtend:=刮板拍照遮光气缸上位 , 
	xPosRetract:= 刮板拍照遮光气缸下位, 
	tTimeout:= T#5S, 
	yValve1=>  刮板拍照遮光气缸, 
	bAlarm=> cyinderAlarm.12);		
//刮板拍照旋转气缸
cylinder_14(
    xManualRetract := , 
    xAutoRetract := , 
    yValve2 => , 
    cylinder_type := 0, 

	xManualAuto:=ManualAuto  , 
	xManualExtend:= 刮板拍照旋转气缸手动 AND 刮板轴9XDATE.fActPos>330, 
	xAutoExtend:=刮板拍照旋转气缸自动 , 
	xReset:=复位  , 
	xPosExtend:=刮板拍照旋转气缸原点  , 
	xPosRetract:= 刮板拍照旋转气缸动点, 
	tTimeout:= T#5S, 
	yValve1=>  刮板拍照旋转气缸   , 
	bAlarm=> cyinderAlarm.13);		
//刮板拍照下压气缸
cylinder_15(
    xManualRetract := , 
    xAutoRetract := , 
    yValve2 => , 
    cylinder_type := 0, 

	xManualAuto:=ManualAuto  , 
	xManualExtend:= 刮板拍照下压气缸手动, 
	xAutoExtend:=刮板拍照下压气缸自动 , 
	xReset:=复位  , 
	xPosExtend:=刮板拍照下压气缸上位, 
	xPosRetract:=刮板拍照下压气缸手动 OR 刮板拍照下压气缸自动 , 
	tTimeout:= T#5S, 
	yValve1=>  刮板拍照下压气缸, 
	bAlarm=> cyinderAlarm.14);
//展缸1进液电池阀1
cylinder_17(
    xManualRetract := , 
    xAutoRetract := , 
    yValve2 => , 
    cylinder_type :=0 , 

	xManualAuto:=ManualAuto  , 
	xManualExtend:= 展缸1进液电池阀1手动, 
	xAutoExtend:= 展缸1进液电池阀1自动, 
	xReset:=复位  , 
	xPosExtend:=   , 
	xPosRetract:= , 
	tTimeout:= , 
	yValve1=> 展缸1进液电池阀1, 
	bAlarm=> );	
//展缸1进液电池阀2
cylinder_18(
    xManualRetract := , 
    xAutoRetract := , 
    yValve2 => , 
    cylinder_type := 0, 

	xManualAuto:=ManualAuto  , 
	xManualExtend:= 展缸1进液电池阀2手动, 
	xAutoExtend:= 展缸1进液电池阀2自动, 
	xReset:=复位  , 
	xPosExtend:=   , 
	xPosRetract:= , 
	tTimeout:= , 
	yValve1=> 展缸1进液电池阀2, 
	bAlarm=> );	
//展缸1进液电池阀3
cylinder_19(
    xManualRetract := , 
    xAutoRetract := , 
    yValve2 => , 
    cylinder_type := 0, 

	xManualAuto:=ManualAuto  , 
	xManualExtend:= 展缸1进液电池阀3手动, 
	xAutoExtend:= 展缸1进液电池阀3自动, 
	xReset:=复位  , 
	xPosExtend:=   , 
	xPosRetract:= , 
	tTimeout:= , 
	yValve1=> 展缸1进液电池阀3, 
	bAlarm=> );	
//展缸1进液电池阀4
cylinder_20(
    xManualRetract := , 
    xAutoRetract := , 
    yValve2 => , 
    cylinder_type := 0, 

	xManualAuto:=ManualAuto  , 
	xManualExtend:= 展缸1进液电池阀4手动, 
	xAutoExtend:= 展缸1进液电池阀4自动, 
	xReset:=复位  , 
	xPosExtend:=   , 
	xPosRetract:= , 
	tTimeout:= , 
	yValve1=> 展缸1进液电池阀4, 
	bAlarm=> );	
//展缸1排液电池阀1
cylinder_21(
    xManualRetract := , 
    xAutoRetract := , 
    yValve2 => , 
    cylinder_type := 0, 

	xManualAuto:=ManualAuto  , 
	xManualExtend:= 展缸1排液电池阀1手动, 
	xAutoExtend:= 展缸1排液电池阀1自动, 
	xReset:=复位  , 
	xPosExtend:=   , 
	xPosRetract:= , 
	tTimeout:= , 
	yValve1=> 展缸1排液电池阀1, 
	bAlarm=> );	
//展缸1排液电池阀2
cylinder_22(
    xManualRetract := , 
    xAutoRetract := , 
    yValve2 => , 
    cylinder_type :=0 , 

	xManualAuto:=ManualAuto  , 
	xManualExtend:= 展缸1排液电池阀2手动, 
	xAutoExtend:= 展缸1排液电池阀2自动, 
	xReset:=复位  , 
	xPosExtend:=   , 
	xPosRetract:= , 
	tTimeout:= , 
	yValve1=> 展缸1排液电池阀2, 
	bAlarm=> );	
//展缸1排液电池阀3
cylinder_23(
    xManualRetract := , 
    xAutoRetract := , 
    yValve2 => , 
    cylinder_type :=0 , 

	xManualAuto:=ManualAuto, 
	xManualExtend:= 展缸1排液电池阀3手动, 
	xAutoExtend:= 展缸1排液电池阀3自动, 
	xReset:=复位  , 
	xPosExtend:=   , 
	xPosRetract:= , 
	tTimeout:= , 
	yValve1=> 展缸1排液电池阀3, 
	bAlarm=> );	
//展缸1排液电池阀4
cylinder_24(
    xManualRetract := , 
    xAutoRetract := , 
    yValve2 => , 
    cylinder_type := 0, 

	xManualAuto:=ManualAuto, 
	xManualExtend:= 展缸1排液电池阀4手动, 
	xAutoExtend:= 展缸1排液电池阀4自动, 
	xReset:=复位  , 
	xPosExtend:=   , 
	xPosRetract:= , 
	tTimeout:= , 
	yValve1=> 展缸1排液电池阀4, 
	bAlarm=> );	
//展缸1吹气电池阀1
cylinder_25(
    xManualRetract := , 
    xAutoRetract := , 
    yValve2 => , 
    cylinder_type := 0, 

	xManualAuto:=ManualAuto, 
	xManualExtend:= 展缸1吹气电池阀1手动, 
	xAutoExtend:= 展缸1吹气电池阀1自动, 
	xReset:=复位  , 
	xPosExtend:=   , 
	xPosRetract:= , 
	tTimeout:= , 
	yValve1=> 展缸1吹气电池阀1, 
	bAlarm=> );	
//展缸1吹气电池阀2
cylinder_26(
    xManualRetract := , 
    xAutoRetract := , 
    yValve2 => , 
    cylinder_type := 0, 

	xManualAuto:=ManualAuto, 
	xManualExtend:= 展缸1吹气电池阀2手动, 
	xAutoExtend:= 展缸1吹气电池阀2自动, 
	xReset:=复位  , 
	xPosExtend:=   , 
	xPosRetract:= , 
	tTimeout:= , 
	yValve1=> 展缸1吹气电池阀2, 
	bAlarm=> );	
//展缸1吹气电池阀3
cylinder_27(
    xManualRetract := , 
    xAutoRetract := , 
    yValve2 => , 
    cylinder_type := 0, 

	xManualAuto:=ManualAuto  , 
	xManualExtend:= 展缸1吹气电池阀3手动, 
	xAutoExtend:= 展缸1吹气电池阀3自动, 
	xReset:=复位  , 
	xPosExtend:=   , 
	xPosRetract:= , 
	tTimeout:= , 
	yValve1=> 展缸1吹气电池阀3, 
	bAlarm=> );	
//展缸1吹气电池阀4
cylinder_28(
    xManualRetract := , 
    xAutoRetract := , 
    yValve2 => , 
    cylinder_type := 0, 

	xManualAuto:=ManualAuto, 
	xManualExtend:= 展缸1吹气电池阀4手动, 
	xAutoExtend:= 展缸1吹气电池阀4自动, 
	xReset:=复位  , 
	xPosExtend:=   , 
	xPosRetract:= , 
	tTimeout:= , 
	yValve1=> 展缸1吹气电池阀4, 
	bAlarm=> );	
//展缸2进液电池阀1
cylinder_29(
    xManualRetract := , 
    xAutoRetract := , 
    yValve2 => , 
    cylinder_type := 0, 

	xManualAuto:=ManualAuto, 
	xManualExtend:= 展缸2进液电池阀1手动, 
	xAutoExtend:= 展缸2进液电池阀1自动, 
	xReset:=复位  , 
	xPosExtend:=   , 
	xPosRetract:= , 
	tTimeout:= , 
	yValve1=> 展缸2进液电池阀1, 
	bAlarm=> );	
//展缸2进液电池阀2
cylinder_30(
    xManualRetract := , 
    xAutoRetract := , 
    yValve2 => , 
    cylinder_type := 0, 

	xManualAuto:=ManualAuto, 
	xManualExtend:= 展缸2进液电池阀2手动, 
	xAutoExtend:= 展缸2进液电池阀2自动, 
	xReset:=复位  , 
	xPosExtend:=   , 
	xPosRetract:= , 
	tTimeout:= , 
	yValve1=> 展缸2进液电池阀2, 
	bAlarm=> );	
//展缸2进液电池阀3
cylinder_31(
    xManualRetract := , 
    xAutoRetract := , 
    yValve2 => , 
    cylinder_type := 0, 

	xManualAuto:=ManualAuto, 
	xManualExtend:= 展缸2进液电池阀3手动, 
	xAutoExtend:= 展缸2进液电池阀3自动, 
	xReset:=复位  , 
	xPosExtend:=   , 
	xPosRetract:= , 
	tTimeout:= , 
	yValve1=> 展缸2进液电池阀3, 
	bAlarm=> );	
//展缸2进液电池阀4
cylinder_32(
    xManualRetract := , 
    xAutoRetract := , 
    yValve2 => , 
    cylinder_type := 0, 

	xManualAuto:=ManualAuto, 
	xManualExtend:= 展缸2进液电池阀4手动, 
	xAutoExtend:= 展缸2进液电池阀4自动, 
	xReset:=复位  , 
	xPosExtend:=   , 
	xPosRetract:= , 
	tTimeout:= , 
	yValve1=> 展缸2进液电池阀4, 
	bAlarm=> );	
//展缸2排液电池阀1
cylinder_33(
    xManualRetract := , 
    xAutoRetract := , 
    yValve2 => , 
    cylinder_type := 0, 

	xManualAuto:=ManualAuto, 
	xManualExtend:= 展缸2排液电池阀1手动, 
	xAutoExtend:= 展缸2排液电池阀1自动, 
	xReset:=复位  , 
	xPosExtend:=   , 
	xPosRetract:= , 
	tTimeout:= , 
	yValve1=> 展缸2排液电池阀1, 
	bAlarm=> );	
//展缸2排液电池阀2
cylinder_34(
    xManualRetract := , 
    xAutoRetract := , 
    yValve2 => , 
    cylinder_type := 0, 

	xManualAuto:=ManualAuto, 
	xManualExtend:= 展缸2排液电池阀2手动, 
	xAutoExtend:= 展缸2排液电池阀2自动, 
	xReset:=复位  , 
	xPosExtend:=   , 
	xPosRetract:= , 
	tTimeout:= , 
	yValve1=> 展缸2排液电池阀2, 
	bAlarm=> );	
//展缸2排液电池阀3
cylinder_35(
    xManualRetract := , 
    xAutoRetract := , 
    yValve2 => , 
    cylinder_type := 0, 

	xManualAuto:=ManualAuto, 
	xManualExtend:= 展缸2排液电池阀3手动, 
	xAutoExtend:= 展缸2排液电池阀3自动, 
	xReset:=复位  , 
	xPosExtend:=   , 
	xPosRetract:= , 
	tTimeout:= , 
	yValve1=> 展缸2排液电池阀3, 
	bAlarm=> );	
//展缸2排液电池阀4
cylinder_36(
    xManualRetract := , 
    xAutoRetract := , 
    yValve2 => , 
    cylinder_type :=0 , 

	xManualAuto:=ManualAuto, 
	xManualExtend:= 展缸2排液电池阀4手动, 
	xAutoExtend:= 展缸2排液电池阀4自动, 
	xReset:=复位  , 
	xPosExtend:=   , 
	xPosRetract:= , 
	tTimeout:= , 
	yValve1=> 展缸2排液电池阀4, 
	bAlarm=> );	
//展缸2吹气电池阀1
cylinder_37(
    xManualRetract := , 
    xAutoRetract := , 
    yValve2 => , 
    cylinder_type := 0, 

	xManualAuto:=ManualAuto, 
	xManualExtend:= 展缸2吹气电池阀1手动, 
	xAutoExtend:= 展缸2吹气电池阀1自动, 
	xReset:=复位  , 
	xPosExtend:=   , 
	xPosRetract:= , 
	tTimeout:= , 
	yValve1=> 展缸2吹气电池阀1, 
	bAlarm=> );	
//展缸2吹气电池阀2
cylinder_38(
    xManualRetract := , 
    xAutoRetract := , 
    yValve2 => , 
    cylinder_type := 0, 

	xManualAuto:=ManualAuto, 
	xManualExtend:= 展缸2吹气电池阀2手动, 
	xAutoExtend:= 展缸2吹气电池阀2自动, 
	xReset:=复位  , 
	xPosExtend:=   , 
	xPosRetract:= , 
	tTimeout:= , 
	yValve1=> 展缸2吹气电池阀2, 
	bAlarm=> );	
//展缸1吹气电池阀3
cylinder_39(
    xManualRetract := , 
    xAutoRetract := , 
    yValve2 => , 
    cylinder_type := 0, 

	xManualAuto:=ManualAuto, 
	xManualExtend:= 展缸2吹气电池阀3手动, 
	xAutoExtend:= 展缸2吹气电池阀3自动, 
	xReset:=复位  , 
	xPosExtend:=   , 
	xPosRetract:= , 
	tTimeout:= , 
	yValve1=> 展缸2吹气电池阀3, 
	bAlarm=> );	
//展缸2吹气电池阀4
cylinder_40(
    xManualRetract := , 
    xAutoRetract := , 
    yValve2 => , 
    cylinder_type := 0, 

	xManualAuto:=ManualAuto, 
	xManualExtend:= 展缸2吹气电池阀4手动, 
	xAutoExtend:= 展缸2吹气电池阀4自动, 
	xReset:=复位  , 
	xPosExtend:=   , 
	xPosRetract:= , 
	tTimeout:= , 
	yValve1=> 展缸2吹气电池阀4, 
	bAlarm=> );	
//收集进液电池阀
cylinder_41(
    xManualRetract := , 
    xAutoRetract := , 
    yValve2 => , 
    cylinder_type := 0, 

	xManualAuto:=ManualAuto, 
	xManualExtend:= 收集进液手动, 
	xAutoExtend:= 收集进液自动, 
	xReset:=复位  , 
	xPosExtend:=   , 
	xPosRetract:= , 
	tTimeout:= , 
	yValve1=> 收集平台进液2通电池阀, 
	bAlarm=> );	
//收集排液电池阀
cylinder_42(
    xManualRetract := , 
    xAutoRetract := , 
    yValve2 => , 
    cylinder_type := 0, 

	xManualAuto:=ManualAuto  , 
	xManualExtend:= 收集排液手动, 
	xAutoExtend:= 收集排液自动, 
	xReset:=复位  , 
	xPosExtend:=   , 
	xPosRetract:= , 
	tTimeout:= , 
	yValve1=> 收集平台排液3通电池阀, 
	bAlarm=> );	
//收集正压排液电池阀
cylinder_43(
    xManualRetract := , 
    xAutoRetract := , 
    yValve2 => , 
    cylinder_type :=0 , 

	xManualAuto:=ManualAuto  , 
	xManualExtend:= 收集正压排液手动, 
	xAutoExtend:= 收集正压排液自动, 
	xReset:=复位  , 
	xPosExtend:=   , 
	xPosRetract:= , 
	tTimeout:= , 
	yValve1=> 收集平台正压排液阀, 
	bAlarm=> );	
//溶液收集瓶定位气缸
cylinder_44(
    xManualRetract := , 
    xAutoRetract := , 
    yValve2 => , 
    cylinder_type := 0, 

	xManualAuto:=ManualAuto  , 
	xManualExtend:= 溶液收集瓶定位手动, 
	xAutoExtend:= 溶液收集瓶定位自动, 
	xReset:=复位  , 
	xPosExtend:=   , 
	xPosRetract:= , 
	tTimeout:= , 
	yValve1=> 溶液收集瓶工位定位气缸, 
	bAlarm=> );	
//上样定位气缸
cylinder_45(
    xManualRetract := , 
    xAutoRetract := , 
    yValve2 => , 
    cylinder_type :=0 , 

	xManualAuto:=ManualAuto  , 
	xManualExtend:= 上样定位手动, 
	xAutoExtend:= 上样定位自动, 
	xReset:=复位  , 
	xPosExtend:=   , 
	xPosRetract:= , 
	tTimeout:= , 
	yValve1=> 上样定位气缸, 
	bAlarm=> );	
//上样点样三通电池阀
cylinder_46(
    xManualRetract := , 
    xAutoRetract := , 
    yValve2 => , 
    cylinder_type :=0 , 

	xManualAuto:=ManualAuto  , 
	xManualExtend:= 上样点样三通电池阀手动, 
	xAutoExtend:= 上样点样三通电池阀自动, 
	xReset:=复位  , 
	xPosExtend:=   , 
	xPosRetract:= , 
	tTimeout:= , 
	yValve1=> 上样点样三通电池阀, 
	bAlarm=> );	
//刮板拍照真空泵
cylinder_46(
    xManualRetract := , 
    xAutoRetract := , 
    yValve2 => , 
    cylinder_type := 0, 

	xManualAuto:=ManualAuto  , 
	xManualExtend:=刮板拍照真空手动 , 
	xAutoExtend:= 刮板拍照真空自动, 
	xReset:=复位  , 
	xPosExtend:=   , 
	xPosRetract:= , 
	tTimeout:= , 
	yValve1=> 刮板拍照真空阀, 
	bAlarm=> );	
//刮板拍照无刷电机
cylinder_47(
    xManualRetract := , 
    xAutoRetract := , 
    yValve2 => , 
    cylinder_type :=0 , 

	xManualAuto:=ManualAuto  , 
	xManualExtend:=刮板拍照无刷电机手动 , 
	xAutoExtend:=刮板拍照无刷电机自动 , 
	xReset:=复位  , 
	xPosExtend:=   , 
	xPosRetract:= , 
	tTimeout:= , 
	yValve1=> 刮板拍照无刷电机, 
	bAlarm=> );	
//刮板拍照定位气缸
cylinder_48(
    xManualRetract := , 
    xAutoRetract := , 
    yValve2 => , 
    cylinder_type :=0 , 

	xManualAuto:=ManualAuto  , 
	xManualExtend:= 刮板拍照定位气缸手动, 
	xAutoExtend:=刮板拍照定位气缸自动 , 
	xReset:=复位  , 
	xPosExtend:=   , 
	xPosRetract:= , 
	tTimeout:= , 
	yValve1=> 刮板拍照定位气缸, 
	bAlarm=> );	
//粉末收集器定位气缸
cylinder_49(
    xManualRetract := , 
    xAutoRetract := , 
    yValve2 => , 
    cylinder_type :=0 , 

	xManualAuto:=ManualAuto  , 
	xManualExtend:= 粉末收集器定位手动, 
	xAutoExtend:= 粉末收集器定位自动, 
	xReset:=复位  , 
	xPosExtend:=   , 
	xPosRetract:= , 
	tTimeout:= , 
	yValve1=> 粉末收集器工位定位气缸, 
	bAlarm=> );	
//上样吹气电池阀
cylinder_50(
    xManualRetract := , 
    xAutoRetract := , 
    yValve2 => , 
    cylinder_type := 0, 

	xManualAuto:=ManualAuto  , 
	xManualExtend:= 上样吹气手动, 
	xAutoExtend:= 上样吹气自动, 
	xReset:=复位  , 
	xPosExtend:=   , 
	xPosRetract:= , 
	tTimeout:= , 
	yValve1=> 上样吹气二通阀, 
	bAlarm=> );

END_PROGRAM

// Device/Application/25_FB_功能块/FB_cylinder
FUNCTION_BLOCK FB_cylinder
VAR_INPUT
    xManualAuto : BOOL := FALSE;  // 手自动模式：FALSE=手动，TRUE=自动
    xManualExtend : BOOL;  // 手动伸出
	// 手动缩回
	xManualRetract: BOOL;
    xAutoExtend : BOOL;  // 自动伸出
	// 自动缩回
	xAutoRetract: BOOL;
    xReset : BOOL;  // 复位按钮
    xPosExtend : BOOL;  // 伸出到位传感器
    xPosRetract : BOOL;  // 缩回到位传感器
    tTimeout : TIME := T#5S;  // 动作超时时间
END_VAR
VAR_OUTPUT
    yValve1 : BOOL;  // 电磁阀1输出：TRUE=伸出，FALSE=缩回
	// 电磁阀2输出：TRUE=伸出，FALSE=缩回
	yValve2: BOOL;
    bAlarm : BOOL;  // 报警输出
END_VAR
VAR
    bEnableCmd1 : BOOL;  // 有效的命令1
	// 有效的命令1
	bEnableCmd2: BOOL;
	tActionTimer: TON;// 动作定时器
END_VAR
VAR_INPUT
	// 气缸类型  0 单控  1双控
	cylinder_type: INT;
END_VAR



CASE cylinder_type OF
	0:     //单控电池阀
		//命令逻辑选择
		IF xManualAuto  THEN
			//自动模式，使用自动命令
			bEnableCmd1 :=xAutoExtend;
			ELSE
			//手动模式，使用手动命令
			bEnableCmd1 :=xManualExtend  ;
		END_IF
		//控制指令
		IF bEnableCmd1 THEN
			//开始伸出
			yValve1:=TRUE;
			ELSE
			//开始缩回
			yValve1 :=FALSE;
		END_IF
		
	
			tActionTimer(IN := (NOT xPosExtend AND NOT yValve1)  OR   (NOT xPosRetract AND yValve1), PT:=tTimeout );
			bAlarm :=tActionTimer .Q;
	
	1:        //双控电池阀
		//命令逻辑选择
		IF xManualAuto  THEN
			//自动模式，使用自动命令
			bEnableCmd1 :=xAutoExtend;
			bEnableCmd2 :=xAutoRetract;
		ELSE
			//手动模式，使用手动命令
			bEnableCmd1 :=xManualExtend;
			bEnableCmd2 :=xManualRetract;
		END_IF
		//伸出控制指令
		IF bEnableCmd1 THEN
			//开始伸出
			yValve1:=TRUE;
			yValve2:=FALSE;
		ELSE 
			yValve1:=FALSE;
		END_IF
		
		IF bEnableCmd2 THEN
			//开始缩回
			yValve2:=TRUE;
			yValve1:=FALSE;
		ELSE 
			yValve2:=FALSE;
		END_IF
		
			tActionTimer(IN := (NOT xPosExtend AND NOT yValve1)  OR   (NOT xPosRetract AND yValve2), PT:=tTimeout );
			bAlarm :=tActionTimer .Q;
		
END_CASE

IF xReset THEN
	bAlarm:=FALSE ;
END_IF

END_FUNCTION_BLOCK

// Device/Application/40_Man/Sample_point_sampling_上样点样
PROGRAM Sample_point_sampling_上样点样
VAR
	初始化step: INT;
	清洗step: INT;
	清洗计数: INT;
	上样准备step: INT;
	放硅胶板STEP: INT;
	吸收液体step: INT;
	TON_0: TON;
	TON_1: TON;
	点样step: INT;
	stepTimer           : TON;       // 步骤内通用定时器（调试期模拟，实机替换为FB完成信号）
    bubbleIndex         : INT;       // Step 20 气泡序列循环索引
    cleanCounter        : INT;       // Step 10 清洗循环计数器
	泵初始化完成: BOOL;
	R_TRIG: ARRAY[1..12] OF R_TRIG;
	N: INT;
	A: INT;
	TON: ARRAY[1..11] OF TON;
	打样伺服移动step: INT;
END_VAR

// ══════════════════════════════════════════════════════════════
// 上样点样流程序列器 — 简化版 v1.0（定时器驱动，无FB依赖）
// ══════════════════════════════════════════════════════════════
// 对应上位机 Stage: spotting（PLC 变量前缀 Sampling）
// 子步 {0, 10, 20, 30, 40, 50, 90}
// 职责：执行上样点样全流程（清洗→气泡准备→放板→吸液→点样）
//
// 简化要点（相较 [pending]plc_spotting.txt v1.6）：
//   - 去掉 pumpCmd FB 依赖：所有泵步骤用 stepTimer 模拟完成
//   - 去掉 System_Ready 全局守卫：调试期无需先执行 System_Init
//   - 去掉 Sampling_init_instructions 工位级泵初始化
//   - 去掉参数校验：范围检查交给上位机
//   - 去掉 latched 变量：直接读全局变量
//   - 去掉 Phase2 传感器逻辑：Step 20 统一定时器推进
//   - 保留六件套 + 全部业务参数名（与上位机 SpottingStage 完全兼容）
//
// 参照 plc_collection.txt（collect 工位）模板编写
// ══════════════════════════════════════════════════════════════
//
// ★★★ PLC工程师注意事项 ★★★
// 本文件为调试期简化版，所有 stepTimer 模拟的位置均为实机集成点。
// 标记说明：
//   TODO【实机集成点】— 需替换为真实 FB/IO 调用的占位
//   TODO【逻辑判断】  — 实机必须增加的条件检查/安全守卫
//   当前 stepTimer PT:=T#5S 仅为模拟延时，实机应替换为实际完成条件
// ══════════════════════════════════════════════════════════════

IF Sampling_X_coordinate>0 THEN 
TON[11](IN:=NOT 上样料架检测1 OR NOT 上样料架检测2,PT:=T#3S);
	IF TON[11].Q THEN
		上样料架报警:=TRUE;
	END_IF
END_IF

// ── 1. 急停联锁（最高优先级）──
// TODO【逻辑判断】实机急停时应额外执行：
//   - 停止当前正在执行的泵指令（pumpCmd_execute := FALSE）
//   - 关闭上样针三通阀（恢复安全位置）
//   - 若 Step 20 正在执行气泡准备，停止补液泵
IF NOT 急停 THEN
    Sampling_Step  := 0;
    Sampling_Done  := FALSE;
    Sampling_Error := TRUE;
    Sampling_Busy  := FALSE;
	初始化step:=0;
	清洗step:=0;
	清洗计数:=0;
	上样准备step:=0;
	放硅胶板STEP:=0;
	吸收液体step:=0;
	打样伺服移动step:=0;
	泵初始化完成:=FALSE;
	N:=0;
	A:=0;
    stepTimer(IN := FALSE, PT := T#0S);
    RETURN;
END_IF

// ── 2. 复位脉冲（用于错误恢复 / 强制清状态）──
// TODO【逻辑判断】实机复位时应额外执行：
//   - 清空 waitingPumpDone 标志
//   - 清空 Sampling_init_instructions（若使用了工位级泵初始化）
IF Sampling_Reset THEN
    Sampling_Step  := 0;
    Sampling_Done  := FALSE;
    Sampling_Error := FALSE;
    Sampling_Busy  := FALSE;
    stepTimer(IN := FALSE, PT := T#0S);
    cleanCounter := 0;
    bubbleIndex  := 0;
    RETURN;
END_IF

// ── 3. Enable=FALSE 时清 Done（次周期复位握手）──
//    上位机收到 Done 后会拉低 Sampling_Enable，本段确保下一周期 Done 自动归零，
//    避免 Done 残留导致 Step 0 误判。
IF NOT Sampling_Enable THEN
    Sampling_Done := FALSE;
END_IF

// ── 4. 派生 Sampling_Busy（写者唯一：本 POU 是唯一写者，禁止他处赋值）──
Sampling_Busy := (Sampling_Step >= 10)
              AND (Sampling_Step <= 80)
              AND (NOT Sampling_Done);

IF MODE_State=1 THEN
	CASE Sampling_Step OF
		0:  // ═══ 空闲：等待 Enable 上升 ═══
        // TODO【逻辑判断】实机应在 Enable 上升时增加以下校验：
        //   - System_Ready = TRUE（全局初始化已完成，见 plc_system_init.txt）
        //   - Sampling_init_instructions 若非空，先执行泵Z初始化指令
        //   - 参数范围校验：clean_count∈[0,100], bubble_count∈[0,16],
        //     Phase2_MaxCycles∈[0,50]，Phase2启用时 phase2_instructions 非空
        //   - 锁存计数值到局部变量（防止PC中途篡改全局变量）

			IF Sampling_Enable AND (NOT Sampling_Done) THEN
				Sampling_Step := 5;
				stepTimer(IN := FALSE, PT := T#0S);  // 复位定时器
			END_IF
		5:
				A00_initialization_初始化();
				IF Sampling_initialization_OK THEN
					Sampling_initialization_OK:=FALSE;
					Sampling_Step:=10;
				END_IF
		10: // ═══ 清洗（消费 Sampling_clean_instructions + Sampling_clean_count）═══
        // TODO【实机集成点】替换 stepTimer 为真实泵 FB 调用：
        //   按 Sampling_clean_count 循环执行 Sampling_clean_instructions 指令
        //   使用 pumpCmd FB 提交指令，等待 pumpCmd_done 后计数+1
        //   循环完成后消费指令字符串，推进到 Step 20
        // TODO【逻辑判断】实机需判断：
        //   - clean_count=0 时直接跳到 Step 20
        //   - pumpCmd_error 时进入 Step 90 故障态
        //   - 使用锁存值 latchedCleanCount 而非全局变量（防PC中途篡改）	
			A10_clean_清洗();
			IF Sampling_Cleaning_OK THEN
				stepTimer(IN := FALSE, PT := T#0S);
				Sampling_Cleaning_OK:=FALSE;
				Sampling_Step := 20;
			END_IF

		20: // ═══ 气泡准备（消费 Sampling_bubble_instructions + bubble_count）═══
        // TODO【实机集成点】替换 stepTimer 为真实泵 FB 调用，需分两阶段：
        //
        //   Phase 1（计数驱动）：逐条执行 Sampling_bubble_instructions[1..bubble_count]
        //     FOR bubbleIndex := 1 TO latchedBubbleCount DO
        //         pumpCmd_cmd := Sampling_bubble_instructions[bubbleIndex];
        //         pumpCmd_execute := TRUE;
        //         等待 pumpCmd_done / pumpCmd_error
        //     END_FOR
        //
        //   Phase 2（传感器驱动补液）：
        //     WHILE NOT Sampling_BubbleSensor AND phase2CycleCount < latchedPhase2Max DO
        //         pumpCmd_cmd := Sampling_phase2_instructions;
        //         pumpCmd_execute := TRUE;
        //         等待 pumpCmd_done → phase2CycleCount := phase2CycleCount + 1;
        //     END_WHILE
        //     若达到 MaxCycles 仍未触发传感器 → Step 90 故障
        //
        //   Phase 1/2 均为空（bubble_count=0 AND Phase2_MaxCycles=0）→ 直接跳到 Step 30
        //
        // TODO【逻辑判断】实机需判断：
        //   - 指令数组中空串守卫：Sampling_bubble_instructions[i]='' → 故障
        //   - Phase2 MaxCycles 安全校验：达到上限未触发传感器 → 传感器可能故障 → Step 90
        //   - Sampling_BubbleSensor 物理输入映射（见 VAR_GLOBAL 中的 TODO）
			
	
				
				
				A30_Sample_preparation_上样准备();
				IF Sampling_preparation_OK THEN
					Sampling_preparation_OK:=FALSE;
					Sampling_Step:=30;
				END_IF
		 30: // ═══ 放硅胶板（机械臂+传感器自治）═══
			// TODO【实机集成点】替换 stepTimer 为真实机械臂 FB 调用：
			//   Place_materials_放硅胶板();  // 机械臂FB，传感器确认到位后自动推进
			// TODO【逻辑判断】实机需判断：
			//   - 机械臂到位传感器确认（替代定时器延时）
			//   - 机械臂超时保护（传感器未触发 → Step 90）
			A20_Place_materials_放硅胶板();
			IF Sampling_Place_materials_OK THEN
				Sampling_Place_materials_OK:=FALSE;
				stepTimer(IN := FALSE, PT := T#0S);
				Sampling_Step := 40;
			END_IF	

		40: // ═══ 吸液（消费 Sampling_X/Y_coordinate + Sampling_aspirate_instructions）═══
			// TODO【实机集成点】替换 stepTimer 为真实 FB 调用：
			//   1. 移动到坐标 (X, Y)：moveCmd 执行，等待到位信号
			//   2. 执行吸液泵指令：pumpCmd_cmd := Sampling_aspirate_instructions;
			//      pumpCmd_execute := TRUE; 等待 pumpCmd_done
			// TODO【逻辑判断】实机需判断：
			//   - 移动到位确认（坐标到达传感器）
			//   - pumpCmd_error 时进入 Step 90
			//   - 移动+吸液需串行化：moveCmd完成 → pumpCmd执行
			A40_absorb_liquid_吸收液体();
			IF Sampling_liquid_absorption THEN
				Sampling_liquid_absorption:=FALSE;
				stepTimer(IN := FALSE, PT := T#0S);
				Sampling_Step := 50;
			END_IF
		50: // ═══ 点样（消费 Sampling_dispense_instructions）═══
			// TODO【实机集成点】替换 stepTimer 为真实泵 FB 调用：
			//   pumpCmd_cmd := Sampling_dispense_instructions;
			//   pumpCmd_execute := TRUE; 等待 pumpCmd_done
			// TODO【逻辑判断】实机需判断：
			//   - pumpCmd_error 时进入 Step 90
			A50_Spray_sample_点样();
			IF Sampling_Spray_sample_OK  THEN
				Sampling_Spray_sample_OK:=FALSE;
				Sampling_Step := 60;
				
			END_IF
		60:
			IF  取点样硅胶板完成 THEN
				取点样硅胶板完成:=FALSE;
				stepTimer(IN := FALSE, PT := T#0S);
				Sampling_Done := TRUE;
				Sampling_Busy := FALSE;
				Sampling_Step := 0;
			END_IF
	
		90: // ═══ 故障态：等待外部 Sampling_Reset 脉冲 ═══
			Sampling_Error := TRUE;   // 故障态本身不动作，仅等待顶部复位逻辑
		

	END_CASE	
END_IF

ACTION A20_Place_materials_放硅胶板:



	CASE 放硅胶板STEP OF
	 	0:
			点样轴7YDATE.fAbsTarget:=HMI_点样轴7Y.position[1];
			点样轴7YDATE.xMoveAbs:=TRUE;
			放硅胶板STEP:=10;
		10:
			IF 点样轴7YDATE.bAbMoveDone THEN
				上样点样允许放硅胶板:=TRUE;
				点样轴7YDATE.xMoveAbs:=FALSE;
				放硅胶板STEP:=20;
			END_IF
		20:
			IF 上样点样放硅胶板完成 THEN
				上样点样允许放硅胶板:=FALSE;
				上样点样放硅胶板完成:=FALSE;
				上样定位自动:=TRUE;
				Sampling_Place_materials_OK:=TRUE;
				放硅胶板STEP:=0;
			END_IF
		
		
	 END_CASE
END_ACTION

ACTION A40_absorb_liquid_吸收液体:
TON_0(IN:=吸收液体step=30, PT:=T#0.5S , Q=> , ET=> );
TON_1(IN:=NOT 点样气泡传感器, PT:=T#5S , Q=> , ET=> );
R_TRIG[10](CLK:=%MX2005.5 , Q=> );  //泵空闲中

IF Sampling_X_coordinate>0 AND  Sampling_Y_coordinate>0  THEN
	CASE 吸收液体step OF
		0:
			上样轴5Z轴DATE.fAbsTarget:=0;
			上样轴5Z轴DATE.xMoveAbs:=TRUE;
			IF 上样轴5Z轴DATE.bAbMoveDone THEN
				上样轴5Z轴DATE.xMoveAbs:=FALSE;
				上样轴4X轴DATE.fAbsTarget:=HMI_上样轴4X轴.position[Sampling_X_coordinate];
				打样瓶上料轴3YDATE.fAbsTarget:=HMI_打样瓶上料轴3Y.position[Sampling_Y_coordinate];
				上样轴4X轴DATE.xMoveAbs:=TRUE;
				打样瓶上料轴3YDATE.xMoveAbs:=TRUE;
				吸收液体step:=10;
			END_IF
		10:
			IF 上样轴4X轴DATE.bAbMoveDone AND 打样瓶上料轴3YDATE.bAbMoveDone THEN
				上样轴4X轴DATE.xMoveAbs:=FALSE;
				打样瓶上料轴3YDATE.xMoveAbs:=FALSE;
				上样轴5Z轴DATE.fAbsTarget:=HMI_上样轴5Z轴.position[2];
				上样轴5Z轴DATE.xMoveAbs:=TRUE;
				吸收液体step:=20;
			END_IF
		20:
			IF 上样轴5Z轴DATE.bAbMoveDone THEN
				上样轴5Z轴DATE.xMoveAbs:=FALSE;
				A:=1;
				吸收液体step:=25;
			END_IF
		25:
			CASE A OF
				1,2:
					IF  %MW1300=0 AND NOT 泵站位符 THEN
						转发转存:=Sampling_sample_instructions[A];   //吸收液体
						%MW1300:=LEN(STR:= 转发转存);
						泵站位符:=TRUE;
						吸收液体step:=30;
					END_IF
			END_CASE
					
		
		30:
			IF  %MW1300=0 AND TON_0.Q THEN                        
				转发转存:='/4Q$R';          //查询泵状态指令
				%MW1300:=LEN(STR:= 转发转存);
				
				IF R_TRIG[10].Q THEN
					泵站位符:=FALSE;
					A:=A+1;
					IF A>2 THEN
						A:=0;
						大真空泵站位[11]:=FALSE;
						吸收液体step:=40;
					ELSE
						吸收液体step:=25;
					END_IF
				END_IF
			END_IF

		40:
			上样轴5Z轴DATE.fAbsTarget:=0;
			上样轴5Z轴DATE.xMoveAbs:=TRUE;
			IF 上样轴5Z轴DATE.bAbMoveDone THEN
				上样轴5Z轴DATE.xMoveAbs:=FALSE;
				Sampling_liquid_absorption:=TRUE;
				吸收液体step:=0;
			END_IF

	END_CASE
END_IF
END_ACTION

ACTION A30_Sample_preparation_上样准备:
TON[2](IN:=上样准备step=2,PT:=T#0.5S);
R_TRIG[3](CLK:=%MX2005.5 , Q=> );  //泵空闲中

CASE 上样准备step OF
	0:
		上样轴5Z轴DATE.fAbsTarget:=0;
		上样轴5Z轴DATE.xMoveAbs:=TRUE;
		IF 上样轴5Z轴DATE.bAbMoveDone THEN
			N:=1;
			上样轴5Z轴DATE.xMoveAbs:=FALSE ;
			上样准备step:=1;
		END_IF
		
	1:
	
		CASE N OF
			1,2:
				IF %MW1300=0 AND NOT 泵站位符 THEN
					泵站位符:=TRUE;
					转发转存:=Sampling_prep_instructions[N];    
					%MW1300:=LEN(STR:= 转发转存);   //发送字节数
					上样准备step:=2;
				END_IF
		END_CASE
		
	2:
		IF %MW1300=0 AND TON[2].Q THEN 
		转发转存:='/4Q$R';          //查询泵状态指令
		%MW1300:=LEN(STR:= 转发转存);
		END_IF
		
		IF R_TRIG[3].Q THEN
			泵站位符:=FALSE;
			N:=N+1;
			IF N>2 THEN
				
				Sampling_preparation_OK:=TRUE;
				N:=0;
				上样准备step:=0;
			ELSE
				上样准备step:=1;
			END_IF
			
		END_IF
END_CASE
END_ACTION

ACTION A10_clean_清洗:
TON[1](IN:=清洗step=20,PT:=T#0.5S);
TON[6](IN:=清洗step=40,PT:=T#0.5S);
TON[8](IN:=清洗step=26,PT:=T#0.5S);
R_TRIG[2](CLK:=%MX2005.5 , Q=> );  //泵空闲中
R_TRIG[11](CLK:=%MX2005.5 , Q=> );  //泵空闲中
R_TRIG[12](CLK:=%MX2005.5 , Q=> );  //泵空闲中

CASE 清洗step OF
	0 :
		点样轴6XDATE.xMoveAbs:=FALSE;
		上样轴4X轴DATE.xMoveAbs:=FALSE;
		上样轴5Z轴DATE.xMoveAbs:=FALSE;
		清洗step:=5;
	5:
		点样轴6XDATE.fAbsTarget:=HMI_点样轴6X.position[1];               //6X清洗位置赋值
		上样轴4X轴DATE.fAbsTarget:=HMI_上样轴4X轴.position[9];           //4X清洗位置赋值
		点样轴6XDATE.xMoveAbs:=TRUE;
		上样轴4X轴DATE.xMoveAbs:=TRUE;
		清洗计数:=0;
		清洗step:=6;
	6:
		IF 上样轴4X轴DATE.bAbMoveDone THEN
			上样轴4X轴DATE.xMoveAbs:=FALSE;
			上样轴5Z轴DATE.fAbsTarget:=HMI_上样轴5Z轴.position[1];
			上样轴5Z轴DATE.xMoveAbs:=TRUE;
			清洗step:=7;
		END_IF

	7:
		IF  上样轴5Z轴DATE.bAbMoveDone AND 点样轴6XDATE.bAbMoveDone THEN
			上样轴5Z轴DATE.xMoveAbs:=FALSE;
			点样轴6XDATE.xMoveAbs:=FALSE;
			IF Sampling_clean_count>0 THEN
				清洗step:=10;
			ELSE
				清洗step:=60;
			END_IF
			
		END_IF
	10:
		IF %MW1300=0 AND NOT 泵站位符 THEN
			泵站位符:=TRUE;
			转发转存:=Sampling_clean_instructions[1];    
			%MW1300:=LEN(STR:= 转发转存);   //发送字节数
			大真空泵站位[11]:=TRUE;
			上样点样三通电池阀自动:=TRUE;
			清洗step:=20;
		END_IF
	20:
		IF %MW1300=0 AND TON[1].Q THEN
		转发转存:='/4Q$R';          //查询泵状态指令
		%MW1300:=LEN(STR:= 转发转存);
		END_IF
		
		IF R_TRIG[2].Q THEN
			上样点样三通电池阀自动:=FALSE;
			泵站位符:=FALSE;
			清洗step:=24;
		END_IF
	24:
		IF %MW1300=0 AND NOT 泵站位符 THEN
			泵站位符:=TRUE;
			转发转存:=Sampling_clean_instructions[1];    
			%MW1300:=LEN(STR:= 转发转存);   //发送字节数
			清洗step:=26;
		END_IF
	26:
		IF %MW1300=0 AND TON[8].Q THEN
		转发转存:='/4Q$R';          //查询泵状态指令
		%MW1300:=LEN(STR:= 转发转存);
		END_IF
		
		IF R_TRIG[11].Q THEN
			
			泵站位符:=FALSE;
			清洗step:=30;
		END_IF
	30:
		IF %MW1300=0 AND NOT 泵站位符 THEN
			泵站位符:=TRUE;
			转发转存:=Sampling_clean_instructions[2];    
			%MW1300:=LEN(STR:= 转发转存);   //发送字节数
			
			清洗step:=40;
		END_IF
				
	40:
		IF %MW1300=0 AND TON[6].Q THEN
		转发转存:='/4Q$R';          //查询泵状态指令
		%MW1300:=LEN(STR:= 转发转存);
		END_IF
		
		IF R_TRIG[12].Q THEN
			泵站位符:=FALSE;
			清洗step:=50;
		END_IF
	50:
		清洗计数:=清洗计数+1;
		IF  Sampling_clean_count> 清洗计数 THEN                 
			转发转存:='';
			%MW1300:=128;
			清洗step:=10;
		ELSIF  Sampling_clean_count<= 清洗计数 THEN
			转发转存:='';
			%MW1300:=128;
			清洗计数:=0;
			Sampling_Cleaning_OK:=TRUE;
			清洗step:=0;
		END_IF	
		上样点样三通电池阀自动:=FALSE;
		
	60:
		大真空泵站位[11]:=FALSE;
		Sampling_Cleaning_OK:=TRUE;
		清洗step:=0;
END_CASE
END_ACTION

ACTION A50_Spray_sample_点样:
TON[4](IN:=点样step=20,PT:=T#0.5S);
TON[5](IN:=点样气泡传感器,PT:=T#5S);
TON[7](IN:=点样step=10,PT:=T#0.5S);
R_TRIG[10](CLK:=%MX2005.5 , Q=> );  //泵空闲中

CASE 点样step OF
	0:
		点样轴6XDATE.xMoveAbs:=FALSE;
		点样轴7YDATE.xMoveAbs:=FALSE;
		点样step:=1;
	1:
		点样轴6XDATE.fAbsTarget:=HMI_点样轴6X.position[2];        //起始位
		点样轴7YDATE.fAbsTarget:=HMI_点样轴7Y.position[2];         //起始位
		点样轴6XDATE.xMoveAbs:=TRUE;
		点样轴7YDATE.xMoveAbs:=TRUE;
		点样step:=5;
	5:
		IF 点样轴6XDATE.bAbMoveDone AND 点样轴7YDATE.bAbMoveDone THEN
			点样轴6XDATE.xMoveAbs:=FALSE;
			点样轴7YDATE.xMoveAbs:=FALSE;
			IF  %MW1300=0 AND NOT 泵站位符 THEN
				
				泵站位符:=TRUE;
				转发转存:=Sampling_dispense_instructions[1];
				%MW1300:=LEN(STR:= 转发转存);
				上样点样三通电池阀自动:=TRUE;
				点样step:=10;
			END_IF
		END_IF
	10:
		IF  %MW1300=0 AND TON[7].Q THEN                        
				转发转存:='/4Q$R';          //查询泵状态指令
				%MW1300:=LEN(STR:= 转发转存);
				
				IF R_TRIG[10].Q THEN
					泵站位符:=FALSE;
					
					点样step:=15;
				END_IF
		END_IF
	15:
		IF  %MW1300=0 AND NOT 泵站位符 THEN
			上样吹气自动:=TRUE;
			泵站位符:=TRUE;
			转发转存:=Sampling_dispense_instructions[2];
			%MW1300:=LEN(STR:= 转发转存);
			点样轴6XDATE.fAbsTarget:=HMI_点样轴6X.position[3];             //终点位
			点样轴6XDATE.xMoveAbs:=TRUE;
			点样step:=20;
		END_IF

	20:
		IF  %MW1300=0 AND TON[4].Q THEN                        
				转发转存:='/4Q$R';          //查询泵状态指令
				%MW1300:=LEN(STR:= 转发转存);
				
				IF R_TRIG[10].Q THEN
					泵站位符:=FALSE;
					上样点样三通电池阀自动:=FALSE;
					上样吹气自动:=FALSE;
				END_IF
		END_IF
		CASE 打样伺服移动step OF
			0:
				IF 点样轴6XDATE.bAbMoveDone THEN
					点样轴6XDATE.xMoveAbs:=FALSE;
					IF 泵站位符 THEN
						打样伺服移动step:=10;
					ELSE
						点样step:=30;
					END_IF
					
				END_IF
			10:
				点样轴6XDATE.fAbsTarget:=HMI_点样轴6X.position[2];        //起始位
				点样轴6XDATE.xMoveAbs:=TRUE;
				打样伺服移动step:=20;
			20:
				IF 点样轴6XDATE.bAbMoveDone THEN
					点样轴6XDATE.xMoveAbs:=FALSE;
					打样伺服移动step:=30;
				END_IF
			30:
				点样轴6XDATE.fAbsTarget:=HMI_点样轴6X.position[3];             //终点位
				点样轴6XDATE.xMoveAbs:=TRUE;
				打样伺服移动step:=0;
				
		END_CASE
		
	30:
		点样轴6XDATE.fAbsTarget:=HMI_点样轴6X.position[1];        //清洗位
		点样轴6XDATE.xMoveAbs:=TRUE;
		IF 点样轴6XDATE.bAbMoveDone THEN
			点样轴7YDATE.fAbsTarget:=HMI_点样轴7Y.position[1]; 
			点样轴7YDATE.xMoveAbs:=TRUE;
		
		点样step:=40;
		END_IF
		
	40:
		IF 点样轴7YDATE.bAbMoveDone  THEN
			点样轴6XDATE.xMoveAbs:=FALSE;
			点样轴7YDATE.xMoveAbs:=FALSE;
			上样定位自动:=FALSE;
			上样点样允许取硅胶板:=TRUE;
			Sampling_Spray_sample_OK:=TRUE;
			点样step:=0;
		END_IF
 END_CASE
END_ACTION

ACTION A00_initialization_初始化:





CASE 初始化step OF
	0 :
		上样定位手动:=FALSE;
		上样定位自动:=FALSE;
		上样点样三通电池阀手动:=FALSE;
		上样点样三通电池阀自动:=FALSE;
		上样吹气手动:=FALSE;
		上样吹气自动:=FALSE;
		打样瓶上料轴3YDATE.fAbsTarget:=0;
		点样轴6XDATE.fAbsTarget:=0;
		点样轴7YDATE.fAbsTarget:=0;
		上样轴4X轴DATE.fAbsTarget:=0;
		上样轴5Z轴DATE.fAbsTarget:=0;
		上样点样允许放硅胶板:=FALSE;
		点样轴7YDATE.xMoveAbs:=FALSE;
		点样轴6XDATE.xMoveAbs:=FALSE;
		上样轴5Z轴DATE.xMoveAbs:=FALSE;
		上样轴4X轴DATE.xMoveAbs:=FALSE;
		打样瓶上料轴3YDATE.xMoveAbs:=FALSE;
		Sampling_Spray_sample_OK:=FALSE;
		Sampling_liquid_absorption:=FALSE;
		Sampling_preparation_OK:=FALSE;
		上样点样允许取硅胶板:=FALSE;
		上样点样放硅胶板完成:=FALSE;
		大真空泵站位[11]:=FALSE;
		清洗计数:=0;
		清洗step:=0;
		放硅胶板STEP:=0;
		上样准备step:=0;
		吸收液体step:=0;
		点样step:=0;
		初始化step:=5;
	5:
		上样轴5Z轴DATE.fAbsTarget:=0;
		上样轴5Z轴DATE.xMoveAbs:=TRUE;
		IF 上样轴5Z轴DATE.bAbMoveDone THEN
			点样轴7YDATE.fAbsTarget:=0  ;  
			点样轴6XDATE.fAbsTarget:=0  ; 
			上样轴4X轴DATE.fAbsTarget:=0;          
			上样轴4X轴DATE.xMoveAbs:=TRUE;
			点样轴7YDATE.xMoveAbs:=TRUE;
			点样轴6XDATE.xMoveAbs:=TRUE;
			初始化step:=6;
		END_IF
	6:
		IF 上样轴4X轴DATE.bAbMoveDone AND 上样轴5Z轴DATE.bAbMoveDone AND 点样轴6XDATE.bAbMoveDone AND 点样轴7YDATE.bAbMoveDone THEN
			初始化step:=10;
			上样轴4X轴DATE.xMoveAbs:=FALSE;
			点样轴7YDATE.xMoveAbs:=FALSE;
			上样轴5Z轴DATE.xMoveAbs:=FALSE;
			点样轴6XDATE.xMoveAbs:=FALSE;
		END_IF
	10:
		IF %MW1300=0 AND NOT 泵站位符 THEN
			泵站位符:=TRUE;
			转发转存:='/4Z0,1,1R$R';     //泵初始化指令 
			%MW1300:=LEN(STR:= 转发转存);   //发送字节数
			初始化STEP:=20;
		END_IF
	20:
		IF %MW1300=0 THEN
			转发转存:='/4Q$R';          //查询泵状态指令
			%MW1300:=LEN(STR:= 转发转存);
		END_IF
		R_TRIG[1](CLK:=%MX2005.5 , Q=> );  //泵空闲中
		IF R_TRIG[1].Q THEN
			泵站位符:=FALSE;
			初始化STEP:=30;
		END_IF
	30:
		
		
			Sampling_initialization_OK:=TRUE;
			初始化step:=0;
		

END_CASE
END_ACTION

END_PROGRAM

// Device/Application/40_Man/Collection_process_收集流程
PROGRAM Collection_process_收集流程
VAR
	准备step: INT;
	收集step: INT;
	TON_0: TON;
	搬运step: INT;
	
	
	ton3s: TON;

	ton5s: TON;
	i: INT;
	
	stepTimer: TON;
	R_TRIG: ARRAY[1..5] OF R_TRIG;
	泵初始化完成: BOOL;
	初始化STEP: INT;
	ton: ARRAY[1..10] OF TON;
END_VAR

// TON自复位：Q变TRUE后IN立即变FALSE，下周期复位，形成循环脉冲
ton3s(IN := bEnable AND NOT ton3s.Q, PT := T#3S);

// Q脉冲时翻转输出（Q仅维持一个周期，无需上升沿检测）
IF ton3s.Q THEN
    bOutput := NOT bOutput;
END_IF

// ── 1. 急停联锁（最高优先级）──
IF NOT 急停 THEN
    collect_Step  := 0;
    collect_Done  := FALSE;
    collect_Error := TRUE;
    collect_Busy  := FALSE;
	准备step:=0;
	收集step:=0;
	搬运step:=0;
	初始化STEP:=0;
	泵初始化完成:=FALSE;
    stepTimer(IN := FALSE, PT := T#0S);
    RETURN;
END_IF

// ── 2. 复位脉冲（用于错误恢复 / 强制清状态）──
IF collect_Reset THEN
    collect_Step  := 0;
    collect_Done  := FALSE;
    collect_Error := FALSE;
    collect_Busy  := FALSE;
    stepTimer(IN := FALSE, PT := T#0S);
    RETURN;
END_IF

// ── 3. Enable=FALSE 时清 Done（次周期复位握手）──
//    上位机收到 Done 后会拉低 collect_Enable，本段确保下一周期 Done 自动归零，
//    避免 Done 残留导致 step 0 误判。
IF NOT collect_Enable THEN
    collect_Done := FALSE;
END_IF

// ── 4. 派生 collect_Busy（写者唯一：本 POU 是唯一写者，禁止他处赋值）──
collect_Busy := (collect_Step >= 10)
                    AND (collect_Step <= 80)
                    AND (NOT collect_Done);






IF MODE_State=1 THEN
	CASE collect_Step OF
		0 :                      // 空闲：等待 Enable 上升
			 IF collect_Enable AND (NOT collect_Done) THEN
				collect_Step := 5;
			 END_IF
		
		5:	
		    A00_initialization_初始化();
			IF 收集平台下压气缸原点 AND 收集平台夹持气缸原点 AND 收集平台升降气缸原点 AND 收集平台推出气缸原点 AND 泵初始化完成 THEN
				collect_Step:=10;
				泵初始化完成:=FALSE;
			END_IF
			
			
				
		10:                    //就位
				A10_preparation_准备();
			IF collect_prepare_OK THEN
				collect_prepare_OK:=FALSE;
				collect_Step:=20;
			END_IF
			
			
			
		20:                    //收集    	
			A20_collect_收集();
			IF collect_OK THEN
				
				FOR i := 1 TO collect_count BY 1 DO
					;   // 占位：单次打液动作（实机替换为真实调用）
				END_FOR
				collect_OK:=FALSE;
				collect_Step:=30;
			END_IF
			
			
		30:                    //物料搬运
			A30_transport_物料搬运();
			 IF 收集工位放收集器完成 THEN
				 收集工位放收集器完成:=FALSE;
				collect_Done := TRUE;
				collect_Step:=0;
			 END_IF	
			 
			 
		90: // 故障：等待外部 collect_Reset 脉冲（已在顶部统一处理）
			collect_Error := TRUE;   // 故障态本身不动作，仅等待复位
	END_CASE
END_IF

ACTION A30_transport_物料搬运:


CASE 搬运step OF
	0 :                     //复位气缸
		收集下压气缸自动:=FALSE;
		
		搬运step:=5;
	5:
		IF 收集平台下压气缸原点 THEN
			收集升降气缸自动:=FALSE;
			搬运step:=10;
		END_IF
	10:                    //复位伸缩气缸
		IF 收集平台升降气缸原点 THEN
			收集伸缩气缸自动:=TRUE;
			搬运step:=20;
		END_IF
	20:                    //允许机器人收集瓶
		IF 收集平台推出气缸动点 THEN
			收集工位允许机器人取收集瓶放暂存工位:=TRUE;
			搬运step:=30;
		END_IF
	30:
		IF 收集工位机器人放收集瓶到暂存工位完成 THEN
			收集工位允许机器人取收集瓶放暂存工位:=FALSE;
			收集工位机器人放收集瓶到暂存工位完成:=FALSE;
			收集伸缩气缸自动:=FALSE;
			收集工位允许取收集器:=TRUE;
			搬运step:=40;
		END_IF
	40:
		IF 收集工位机器人到达收集器位置 THEN
				收集工位机器人到达收集器位置:=FALSE;
			收集夹持气缸自动:=FALSE;
			收集工位允许取收集器:=FALSE;
			搬运step:=50;
		END_IF
	50:
		IF 收集平台夹持气缸原点 THEN
			收集工位机器人取收集器放回暂存工位:=TRUE;
			搬运step:=60;
		END_IF
	60:
		 IF 收集工位放收集器完成 THEN
		 	搬运step:=0;
		 END_IF
		
		
		

END_CASE
END_ACTION

ACTION A10_preparation_准备:
//准备工作
CASE 准备step OF	
	0:
		IF 收集平台夹持气缸原点 AND 收集平台下压气缸原点 THEN
		收集工位允许放收集器:=TRUE;
		准备step:=10;
		END_IF
	10:
		IF 收集工位放收集器到工位 THEN
			收集夹持气缸自动:=TRUE;
			收集工位允许放收集器:=FALSE;
			准备step:=20;
		END_IF
	20:
		IF 收集平台夹持气缸动点 THEN
			收集工位允许机器人退出工位:=TRUE;
			准备step:=30;
		END_IF
		
	30:
		IF 收集工位机器人退出完成 THEN
			
			收集工位机器人退出完成:=FALSE;
			收集工位允许机器人退出工位:=FALSE;
			准备step:=40;
		END_IF
	40 :
		IF 收集平台推出气缸原点 AND NOT 收集平台瓶子有无传感器 THEN
			收集伸缩气缸自动:=TRUE;
			准备step:=50;
		END_IF
	50:
		IF 收集平台推出气缸动点 THEN
			收集工位允许放收集瓶:=TRUE;
			准备step:=60;
		END_IF
	60:
	    IF 收集工位放收集瓶完成 THEN
	    	收集工位允许放收集瓶:=FALSE;
			收集工位放收集瓶完成:=FALSE;
			收集伸缩气缸自动:=FALSE;
			准备step:=70;
	    END_IF
	70:
		IF 收集平台推出气缸原点 AND 收集平台瓶子有无传感器 THEN
			收集升降气缸自动:=TRUE;
			准备step:=80;
		ELSIF 收集平台推出气缸原点 AND NOT 收集平台瓶子有无传感器 THEN
			收集伸缩气缸自动:=FALSE;
			准备step:=40;
		END_IF

	80:
		IF 收集平台升降气缸动点  THEN
			收集下压气缸自动:=TRUE;
			collect_prepare_OK:=TRUE;
			准备step:=0;
		END_IF
		
END_CASE
END_ACTION

ACTION A00_initialization_初始化:
R_TRIG[1](CLK:=%MX2005.5 , Q=> );  //泵空闲中

//初始化流程
CASE 初始化STEP OF
	0:
		收集下压气缸手动:=FALSE;
		收集下压气缸自动:=FALSE;
		收集夹持气缸手动:=FALSE;
		收集夹持气缸自动:=FALSE;
		收集升降气缸手动:=FALSE;
		收集升降气缸自动:=FALSE;
		收集伸缩气缸手动:=FALSE;
		收集伸缩气缸自动:=FALSE;
		收集进液手动:=FALSE;
		收集进液自动:=FALSE;
		收集排液手动:=FALSE;
		收集排液自动:=FALSE;
		收集正压排液手动:=FALSE;
		收集正压排液自动:=FALSE;
		溶液收集瓶定位手动:=FALSE;
		收集工位允许放收集瓶:=FALSE;
		收集工位允许放收集器:=FALSE;
		收集工位允许机器人退出工位:=FALSE;
		收集工位允许机器人取收集瓶放暂存工位:=FALSE;
		收集工位允许取收集器:=FALSE;
		收集工位机器人取收集器放回暂存工位:=FALSE;
		
	
		收集工位放收集瓶完成:=FALSE;
		收集工位放收集器到工位:=FALSE;
	
		收集工位机器人退出完成:=FALSE;
		
		收集工位机器人放收集瓶到暂存工位完成:=FALSE;
		
		收集工位机器人到达收集器位置:=FALSE;

		collect_prepare_OK:=FALSE;
		collect_OK:=FALSE;
		收集工位放收集器完成:=FALSE;
		收集step:=0;
		准备step:=0;
		搬运step:=0;
		IF %MW1300=0 AND NOT 泵站位符 THEN
			泵站位符:=TRUE;
			转发转存:='/3Z0,2,2R$R';     //泵初始化指令 
			%MW1300:=LEN(STR:= 转发转存);   //发送字节数
			初始化STEP:=10;
		END_IF
	10:
		IF %MW1300=0 THEN
			转发转存:='/3Q$R';          //查询泵状态指令
			%MW1300:=LEN(STR:= 转发转存);
		END_IF
		
		IF R_TRIG[1].Q THEN
			泵站位符:=FALSE;
			泵初始化完成:=TRUE;
			初始化STEP:=0;
		END_IF
END_CASE
END_ACTION

ACTION A20_collect_收集:
ton[1](IN:=收集step=10,PT:=T#0.5S);
ton[2](IN:=收集step=30,PT:=T#10S);
R_TRIG[5](CLK:=%MX2005.5 , Q=> );  //泵空闲中
CASE 收集step OF
	0 :
		IF collect_forward_instructions<>'' THEN
			收集进液自动:=TRUE;
			
			
		END_IF
		IF %MW1300=0 AND 泵站位符=FALSE  THEN
			转发转存:=collect_forward_instructions; 
			%MW1300:=LEN(STR:= 转发转存);   //发送字节数
			泵站位符:=TRUE;
			收集step:=10;
		END_IF
	10:
		IF %MW1300=0 AND ton[1].Q THEN
			转发转存:='/3Q$R';          //查询泵状态指令
			%MW1300:=LEN(STR:= 转发转存);
		END_IF
		
		
		IF R_TRIG[5].Q THEN
			泵站位符:=FALSE;
			收集step:=20;
		END_IF
	

	20:
		IF TRUE  THEN    //注射泵完成//
			转发转存:='';
			%MW300:=128;
			收集进液自动:=FALSE;
			收集排液自动:=TRUE;
			收集正压排液自动:=TRUE;
			收集计数:=收集计数+1;
			收集step:=30;
		END_IF
	30:
		IF ton[2].Q THEN
			TON_0(IN:=TRUE, PT:=T#5S , Q=> , ET=> );
			IF 收集计数>=collect_count AND TON_0.Q THEN
				收集计数:=0;
				收集step:=40;
			ELSE
				收集排液自动:=FALSE;
				收集正压排液自动:=FALSE;
				收集step:=0;
			END_IF
		END_IF
	40:
		
			收集排液自动:=FALSE;
			收集正压排液自动:=FALSE;
			collect_OK:=TRUE;
			收集step:=0;

		

		
END_CASE
END_ACTION

END_PROGRAM

// Device/Application/40_Man/Expand_process_展开流程
PROGRAM Expand_process_展开流程
VAR
	清洗STEP: INT;
	TON_0: TON;
	润洗展缸STEP: INT;
	TON_1: TON;
	TON_2: TON;
	上液step: INT;
	放硅胶板step: INT;
	展开step: INT;
	TON_3: TON;
	TON_4: TON;
	stepTimer   : TON;       // 步骤内通用定时器
    targetTank  : INT;       // 本轮 prep 的目标缸号（锁存值）
    targetGroup : INT;       // 推导的组号（1 或 2）
    targetNum   : INT;       // 推导的组内序号（1-4）
    i           : INT;       // 循环索引
	
	ton3s: TON;
	初始化step: INT;
	泵初始化完成: BOOL;
	R_TRIG: ARRAY[1..10] OF R_TRIG;
	TON: ARRAY[1..10] OF TON;
	润洗计数: INT;
	上液计数: INT;
END_VAR

// ══════════════════════════════════════════════════════════════
// 展开工位准备序列器（协议 v1.2+ / Phase MultiTank）
// ══════════════════════════════════════════════════════════════
// 对应上位机 Stage: develop（PLC 变量前缀 Expand）
// 子步 {0, 10, 20, 30, 40, 90}
// 职责：执行 prep 流程（润洗→上液→放板→交付至展开态）
// 语义变更：Expand_Done = prep完成（非整流程完成）
// 序列器释放后可立即接受下一个 prep 请求
// 排液由独立程序 PRG_TankDrain 处理（见 develop_tank_drain.txt）
//
// 参照 plc_collection.txt（collect 工位）模板编写
// ══════════════════════════════════════════════════════════════

IF 大真空泵站位[0] OR 大真空泵站位[1] OR 大真空泵站位[2] OR 大真空泵站位[3] OR 大真空泵站位[4] OR 大真空泵站位[5] OR 大真空泵站位[6] OR 大真空泵站位[7] OR 大真空泵站位[8] OR 大真空泵站位[9] OR 大真空泵站位[10] OR 大真空泵站位[11] THEN
	大真空泵自动:=TRUE;
	ELSE
	大真空泵自动:=FALSE;
END_IF




// ── 1. 急停联锁（最高优先级）──
IF NOT 急停 THEN
    Expand_Step  := 0;
    Expand_Done  := FALSE;
    Expand_Error := TRUE;
    Expand_Busy  := FALSE;
	大真空泵站位[1]:=FALSE;
	大真空泵站位[2]:=FALSE;
	大真空泵站位[3]:=FALSE;
	大真空泵站位[4]:=FALSE;
	大真空泵站位[5]:=FALSE;
	大真空泵站位[6]:=FALSE;
	大真空泵站位[7]:=FALSE;
	大真空泵站位[8]:=FALSE;
	清洗STEP:=0;
	润洗展缸STEP:=0;
	上液step:=0;
	放硅胶板step:=0;
	展开step:=0;
	初始化step:=0;
	泵初始化完成:=FALSE;
	润洗计数:=0;
	上液计数:=0;
    // 急停时将所有 Prepping 状态的缸标记为 Error
    FOR i := 1 TO 8 DO
        IF Tank_State[i] = 10 THEN
            Tank_State[i] := 90;
        END_IF
    END_FOR
    stepTimer(IN := FALSE, PT := T#0S);
    RETURN;
END_IF

// ── 2. 复位脉冲（用于错误恢复 / 强制清状态）──
IF Expand_Reset THEN
    // 清序列器自身状态
    Expand_Step  := 0;
    Expand_Done  := FALSE;
    Expand_Error := FALSE;
    Expand_Busy  := FALSE;
    stepTimer(IN := FALSE, PT := T#0S);
    // 若有活跃 prep 目标缸，将其标记为 Error（避免孤儿缸）
    IF targetTank >= 1 AND targetTank <= 8 THEN
        IF Tank_State[targetTank] = 10 THEN
            Tank_State[targetTank] := 90;
        END_IF
    END_IF
    // 注：Tank_State[90] 的缸由 PC 写 0 复位（ResourceManager.release()）
    RETURN;
END_IF

// ── 3. Enable=FALSE 时清 Done（次周期复位握手）──
IF NOT Expand_Enable THEN
    Expand_Done := FALSE;
END_IF


// ── 4. 派生 Expand_Busy（写者唯一：本 POU 是唯一写者，禁止他处赋值）──
Expand_Busy := (Expand_Step >= 10)
              AND (Expand_Step <= 80)
              AND (NOT Expand_Done);






IF MODE_State=1 THEN	
	CASE Expand_Step OF
		0:  // ═══ 空闲：等待 Enable 上升 ═══
			IF Expand_Enable AND (NOT Expand_Done) THEN
				// 读取目标缸号并校验
				targetTank := Expand_Target_Tank;
	
				// 校验：目标缸号必须在 1-8 范围内
				IF targetTank < 1 OR targetTank > 8 THEN
					Expand_Error := TRUE;
					Expand_Step := 90;
				// 校验：目标缸必须处于 Idle 状态（防止重复 prep）
				ELSIF Tank_State[targetTank] <> 0 THEN
					Expand_Error := TRUE;
					Expand_Step := 90;
				ELSE
					// 自动推导 Group 和 Number
					targetGroup := (targetTank - 1) / 4 + 1;   // 1-4→Group1, 5-8→Group2
					targetNum   := (targetTank - 1) MOD 4 + 1; // 组内序号 1-4
	
					// 写入协议变量（供 FB 调用使用）
					Expand_Group  := targetGroup;
					Expand_Number := targetNum;
	
					// 标记目标缸进入 Prepping 状态
					Tank_State[targetTank] := 10;
	
					// 推进到 Step 10
					Expand_Step := 5;
					stepTimer(IN := FALSE, PT := T#0S);  // 复位定时器
				END_IF
			END_IF
		 5:                //初始化
			
				A00_initialization_初始化();
				IF  泵初始化完成 THEN
					
					泵初始化完成:=FALSE;
					Expand_Step:=10;
				END_IF
		10: // ═══ 润洗/清洗（Expand_Mode_Flag=0→缸模式；=1→管路模式）═══
			// 润洗/清洗操作针对 targetTank 对应的泵组
	// 				IF Expand_Mode_Flag = 0 THEN
	// 					// 缸模式润洗：使用 targetGroup 对应的泵执行润洗
	// 					clean_expand_润洗展缸();     // FB 内部使用 Expand_Group/Number
	// 				ELSIF Expand_Mode_Flag = 1 THEN
	// 					// 管路模式清洗
	// 					pipeline_cleaning_清洗管路(); // FB 内部使用 Expand_Group/Number
	// 				END_IF
			// TODO【实机集成点】替换上方为真实 FB 调用，按完成信号推进
			IF Expand_Mode_Flag=0  THEN
				A20_clean_expand_润洗展缸();
			ELSIF Expand_Mode_Flag=1 THEN
				A10_pipeline_cleaning_清洗管路();
			END_IF
			IF Expand_Group_clean_OK THEN
				Expand_Group_clean_OK:=FALSE;
				Expand_Step:=20;
			END_IF
		 20: // ═══ 上液（展开剂加入目标展缸）═══
			// 使用 Expand_forward_instructions 中的 DT 协议指令驱动注射泵
			// 目标缸由 targetGroup/targetNum 确定
	//         	up_liquid_上液();    // FB 内部使用 Expand_Group/Number 和 forward_instructions
			// TODO【实机集成点】替换为真实 FB 调用
			IF Expand_Group>0 AND Expand_Number>0 THEN
				A40_up_liquid_上液();
			END_IF
			IF Expand_up_liquid_OK THEN
				Expand_up_liquid_OK:=FALSE;
				Expand_Step:=30;
			END_IF
		30: // ═══ 放硅胶板（机械臂+传感器自治）═══
			// 放板由机械臂执行，传感器确认到位后 PLC 自动推进
			// 不再需要 PC 握手确认（旧 Step 35 已废弃）
	//         	silica_gel_plate_放硅胶板();
			// TODO【实机集成点】替换为真实 FB 调用，以传感器到位信号作为完成条件
			A30_silica_gel_plate_放硅胶板();
			IF Expand_silica_gel_plate_OK THEN
				Expand_silica_gel_plate_OK:=FALSE;
				Expand_Step:=40;
			END_IF
	
		40: // ═══ 【关键变更】交付至展开态 —— 立即释放序列器 ═══
			// 旧逻辑：在此等待展开+排液完成后才 Done
			// 新逻辑：设 Tank_State=40 后立即 Done，释放序列器给下一个 prep
	
			// 将目标缸状态从 Prepping(10) 推进到 Developing(40)
			Tank_State[targetTank] := 40;
	
			// 标记 prep 完成，释放序列器
			Expand_Done := TRUE;
			Expand_Busy := FALSE;
			Expand_Step := 0;
	
			// 序列器已归零，可接受下一个 prep 请求
			// 实际展开由缸自身"静置"完成，排液由独立子程序 PRG_TankDrain 处理
	
		90: // ═══ 故障态：等待外部 Expand_Reset 脉冲 ═══
			Expand_Error := TRUE;   // 故障态本身不动作，仅等待顶部复位逻辑
			
			
			


			
	
	
	END_CASE
END_IF

ACTION A20_clean_expand_润洗展缸:
TON[1](IN:=润洗展缸STEP=15,PT:=T#0.1S);
TON_1(IN:= 润洗展缸STEP=20  , PT:=T#5S , Q=> , ET=> );
TON_2(IN:=润洗展缸STEP=30, PT:=T#3S, Q=> , ET=> );
TON[4](IN:=润洗展缸STEP=40,PT:=T#30S);
TON[10](IN:=(Expand_Group=1 AND  展缸1溶剂废液检测传感器) OR (Expand_Group=2 AND  展缸2溶剂废液检测传感器),PT:=T#10S);
R_TRIG[3](CLK:=%MX2005.5 , Q=> );  //泵空闲中



CASE 润洗展缸STEP OF
	0 :
		润洗计数:=0;
		CASE Expand_Group OF
			1:
				CASE Expand_Number OF
					1:
						展缸1进液电池阀1自动:=TRUE;
						展缸1排液电池阀1自动:=TRUE;
						展缸1气缸1自动:=TRUE;
						润洗展缸STEP:=10;
					2:
						展缸1进液电池阀2自动:=TRUE;
						展缸1排液电池阀2自动:=TRUE;
						展缸1气缸2自动:=TRUE;
						润洗展缸STEP:=10;
					3:
						展缸1进液电池阀3自动:=TRUE;
						展缸1排液电池阀3自动:=TRUE;
						展缸1气缸3自动:=TRUE;
						润洗展缸STEP:=10;
					4:
						展缸1进液电池阀4自动:=TRUE;
						展缸1排液电池阀4自动:=TRUE;
						展缸1气缸4自动:=TRUE;
						润洗展缸STEP:=10;
				END_CASE
			
			2:
				CASE Expand_Number OF
					1:
						展缸2进液电池阀1自动:=TRUE;
						展缸2排液电池阀1自动:=TRUE;
						展缸2气缸1自动:=TRUE;
						润洗展缸STEP:=10;
					2:
						展缸2进液电池阀2自动:=TRUE;
						展缸2排液电池阀2自动:=TRUE;
						展缸2气缸2自动:=TRUE;
						润洗展缸STEP:=10;
					3:
						展缸2进液电池阀3自动:=TRUE;
						展缸2排液电池阀3自动:=TRUE;
						展缸2气缸3自动:=TRUE;
						润洗展缸STEP:=10;
					4:
						展缸2进液电池阀4自动:=TRUE;
						展缸2排液电池阀4自动:=TRUE;
						展缸2气缸4自动:=TRUE;
						润洗展缸STEP:=10;
				END_CASE
		END_CASE
	10:		
		IF %MW1300=0 AND 泵站位符=FALSE  THEN
			转发转存:=Expand_forward_instructions;   
			%MW1300:=LEN(STR:= 转发转存);   //发送字节数
			泵站位符:=TRUE;
			润洗展缸STEP:=15;
		END_IF
	15:
		
		IF %MW1300=0 AND TON[1].Q THEN
			CASE Expand_Group OF
				1:
					转发转存:='/1Q$R';           //查询泵状态指令
				2:
					转发转存:='/2Q$R';           //查询泵状态指令
			END_CASE
			%MW1300:=LEN(STR:= 转发转存);
		END_IF
		
		IF R_TRIG[3].Q THEN
			泵站位符:=FALSE;
			润洗计数:=润洗计数+1;
			IF 润洗计数>=Expand_rinse_count THEN
				润洗计数:=0;
				润洗展缸STEP:=20;
			ELSE
				润洗展缸STEP:=10;
			END_IF
			
		END_IF
		
	20:
		//TON_1(IN:= TRUE  , PT:=T#5S , Q=> , ET=> );
		IF TON_1.Q THEN
			转发转存:='';    
			%MW1300:=128;
			润洗展缸STEP:=30;
		END_IF
	30:
		//TON_2(IN:=TRUE, PT:=T#2S, Q=> , ET=> );
		IF TON_2.Q THEN
			大真空泵站位[9]:=TRUE;
			IF TON[10].Q THEN
				
				CASE Expand_Group OF
					1:
						CASE Expand_Number OF
							1:
								展缸1进液电池阀1自动:=FALSE;
								
								展缸1吹气电池阀1自动:=TRUE;
								
								
								润洗展缸STEP:=40;
							2:
								展缸1进液电池阀2自动:=FALSE;
								
								展缸1吹气电池阀2自动:=TRUE;
								
								
								润洗展缸STEP:=40;
							3:
								展缸1进液电池阀3自动:=FALSE;
								
								展缸1吹气电池阀3自动:=TRUE;
								
								
								润洗展缸STEP:=40;
							4:
								展缸1进液电池阀4自动:=FALSE;
								
								展缸1吹气电池阀4自动:=TRUE;
								
								润洗展缸STEP:=40;
						END_CASE
					
					2:
						CASE Expand_Number OF
							1:
								展缸2进液电池阀1自动:=FALSE;
								
								展缸2吹气电池阀1自动:=TRUE;
								
								润洗展缸STEP:=40;
							2:
								展缸2进液电池阀2自动:=FALSE;
								
								展缸2吹气电池阀2自动:=TRUE;
								
								润洗展缸STEP:=40;
							3:
								展缸2进液电池阀3自动:=FALSE;
								
								展缸2吹气电池阀3自动:=TRUE;
								
								润洗展缸STEP:=40;
							4:
								展缸2进液电池阀4自动:=FALSE;
								
								展缸2吹气电池阀4自动:=TRUE;
								润洗展缸STEP:=40;
						END_CASE
				END_CASE
			END_IF
		END_IF
	40:
		IF TON[4].Q THEN
			大真空泵站位[9]:=FALSE;
			CASE Expand_Group OF
				1:
					CASE Expand_Number OF
						1:
							展缸1排液电池阀1自动:=FALSE;
							展缸1吹气电池阀1自动:=FALSE;
							
							Expand_Group_clean_OK:=TRUE;
							润洗展缸STEP:=0;
						2:
							展缸1排液电池阀2自动:=FALSE;
							展缸1吹气电池阀2自动:=FALSE;
							
							Expand_Group_clean_OK:=TRUE;
							润洗展缸STEP:=0;
						3:
							展缸1排液电池阀3自动:=FALSE;
							展缸1吹气电池阀3自动:=FALSE;
							
							Expand_Group_clean_OK:=TRUE;
							润洗展缸STEP:=0;
						4:
							展缸1排液电池阀4自动:=FALSE;
							
							展缸1吹气电池阀4自动:=FALSE;
							Expand_Group_clean_OK:=TRUE;
							润洗展缸STEP:=0;
					END_CASE
				
				2:
					CASE Expand_Number OF
						1:
							展缸2排液电池阀1自动:=FALSE;
							展缸2吹气电池阀1自动:=FALSE;
							
							Expand_Group_clean_OK:=TRUE;
							润洗展缸STEP:=0;
						2:
							展缸2排液电池阀2自动:=FALSE;
							展缸2吹气电池阀2自动:=FALSE;
							
							Expand_Group_clean_OK:=TRUE;
							润洗展缸STEP:=0;
						3:
							展缸2排液电池阀2自动:=FALSE;
							展缸2吹气电池阀3自动:=FALSE;
							
							Expand_Group_clean_OK:=TRUE;
							润洗展缸STEP:=0;
						4:
							展缸2排液电池阀2自动:=FALSE;
							展缸2吹气电池阀4自动:=FALSE;
							
							Expand_Group_clean_OK:=TRUE;
							润洗展缸STEP:=0;
					END_CASE
			END_CASE
		END_IF
END_CASE
END_ACTION

ACTION A30_silica_gel_plate_放硅胶板:



CASE 放硅胶板step OF
	0:
		
		放硅胶板step:=10;
	10:
		展开工位允许放硅胶板1:=TRUE;
		IF 展开工位机器人到达准备点 THEN
			CASE Expand_Group OF
				1:
					CASE Expand_Number OF
						1:
							展缸1气缸1自动:=FALSE;
							IF 展缸1气缸1原点 THEN
								展开工位允许放硅胶板:=TRUE;
								ParameterList1:=1;
								放硅胶板step:=20;
							END_IF
							
						2:
							展缸1气缸2自动:=FALSE;
							IF 展缸1气缸2原点 THEN
								ParameterList1:=2;
								展开工位允许放硅胶板:=TRUE;
								放硅胶板step:=20;
							END_IF
						3:
							展缸1气缸3自动:=FALSE;
							IF 展缸1气缸3原点 THEN
								ParameterList1:=3;
								展开工位允许放硅胶板:=TRUE;
								放硅胶板step:=20;
							END_IF
						4:
							展缸1气缸4自动:=FALSE;
							IF 展缸1气缸4原点 THEN
								ParameterList1:=4;
								展开工位允许放硅胶板:=TRUE;
								放硅胶板step:=20;
							END_IF
					END_CASE
				2:
					CASE Expand_Number OF
						1:
							展缸2气缸1自动:=FALSE;
							IF 展缸2气缸1原点 THEN
								ParameterList1:=5;
								展开工位允许放硅胶板:=TRUE;
								放硅胶板step:=20;
							END_IF
						2:
							展缸2气缸2自动:=FALSE;
							IF 展缸2气缸2原点 THEN
								ParameterList1:=6;
								展开工位允许放硅胶板:=TRUE;
								放硅胶板step:=20;
							END_IF
						3:
							展缸2气缸3自动:=FALSE;
							IF 展缸2气缸3原点 THEN
								ParameterList1:=7;
								展开工位允许放硅胶板:=TRUE;
								放硅胶板step:=20;
							END_IF
						4:
							展缸2气缸4自动:=FALSE;
							IF 展缸2气缸4原点 THEN
								ParameterList1:=8;
								展开工位允许放硅胶板:=TRUE;
								放硅胶板step:=20;
							END_IF
					END_CASE
			END_CASE	
		END_IF
	20:
		IF 展开工位机器人放硅胶板完成 THEN
			展开工位允许放硅胶板:=FALSE;
			展开工位允许放硅胶板1:=FALSE;
			CASE Expand_Group OF
				1:
					CASE Expand_Number OF
						1:
							展缸1气缸1自动:=TRUE ;
							IF 展缸1气缸1动点 THEN
								放硅胶板step:=30;
							END_IF
							
						2:
							展缸1气缸2自动:=TRUE;
							IF 展缸1气缸2动点 THEN
								
								放硅胶板step:=30;
							END_IF
						3:
							展缸1气缸3自动:=TRUE;
							IF 展缸1气缸3动点 THEN
								
								放硅胶板step:=30;
							END_IF
						4:
							展缸1气缸4自动:=TRUE ;
							IF 展缸1气缸4动点 THEN
								
								放硅胶板step:=30;
							END_IF
					END_CASE
				2:
					CASE Expand_Number OF
						1:
							展缸2气缸1自动:=TRUE;
							IF 展缸2气缸1动点 THEN
								
								放硅胶板step:=30;
							END_IF
						2:
							展缸2气缸2自动:=TRUE ;
							IF 展缸2气缸2动点 THEN
								
								放硅胶板step:=30;
							END_IF
						3:
							展缸2气缸3自动:=TRUE;
							IF 展缸2气缸3动点 THEN
								
								放硅胶板step:=30;
							END_IF
						4:
							展缸2气缸4自动:=TRUE;
							IF 展缸2气缸4动点 THEN
								
								放硅胶板step:=30;
							END_IF
					END_CASE
			END_CASE	
		END_IF
	30:
		展开工位机器人放硅胶板完成:=FALSE;
		Expand_silica_gel_plate_OK:=TRUE;
		放硅胶板step:=0;
	
	
	

END_CASE
END_ACTION

ACTION A40_up_liquid_上液:
R_TRIG[6](CLK:=%MX2005.5 , Q=> );  //泵空闲中
TON[9](IN:=上液step=20,PT:=T#0.5S,);
IF Expand_Group>0 AND Expand_Number>0 THEN
	CASE 上液step OF
		0:
			CASE Expand_Group OF
				1:
					CASE Expand_Number OF
						1:
							展缸1进液电池阀1自动:=TRUE;
							上液step:=10;
						2:
							展缸1进液电池阀2自动:=TRUE;
							上液step:=10;
						3:
							展缸1进液电池阀3自动:=TRUE;
							上液step:=10;
						4:
							展缸1进液电池阀4自动:=TRUE;
							上液step:=10;
					END_CASE
				2:
					CASE Expand_Number OF
						1:
							展缸2进液电池阀1自动:=TRUE;
							上液step:=10;
						2:
							展缸2进液电池阀2自动:=TRUE;
							上液step:=10;
						3:
							展缸2进液电池阀3自动:=TRUE;
							上液step:=10;
						4:
							展缸2进液电池阀4自动:=TRUE;
							上液step:=10;
					END_CASE
			END_CASE
		10:
			IF %MW1300=0 AND 泵站位符=FALSE  THEN
				转发转存:=Expand_forward_instructions; 
				%MW1300:=LEN(STR:= 转发转存);   //发送字节数
				泵站位符:=TRUE;
				上液step:=20;
			END_IF
		20:
		
			IF %MW1300=0 AND TON[9].Q  THEN
				CASE Expand_Group OF
					 1:
						 转发转存:='/1Q$R';          //查询泵状态指令
					 2:
						 转发转存:='/2Q$R';          //查询泵状态指令
				END_CASE
				%MW1300:=LEN(STR:= 转发转存);
			END_IF
			
			
			IF R_TRIG[6].Q THEN
				泵站位符:=FALSE;
				转发转存:='';
				%MW1300:=128;
				上液计数:=上液计数+1;
				IF 上液计数>=Expand_up_liquid_count THEN
					上液计数:=0;
					CASE Expand_Group OF
						1:
							CASE Expand_Number OF
								1:
									展缸1进液电池阀1自动:=FALSE;
									;
								2:
									展缸1进液电池阀2自动:=FALSE;
									
								3:
									展缸1进液电池阀3自动:=FALSE;
									
								4:
									展缸1进液电池阀4自动:=FALSE;
									
							END_CASE
						2:
							CASE Expand_Number OF
								1:
									展缸2进液电池阀1自动:=FALSE;
									
								2:
									展缸2进液电池阀2自动:=FALSE;
									
								3:
									展缸2进液电池阀3自动:=FALSE;
									
								4:
									展缸2进液电池阀4自动:=FALSE;
									
							END_CASE
						END_CASE
					Expand_up_liquid_OK:=TRUE;
					上液step:=0;
				ELSE
					上液step:=10;
				END_IF
			END_IF	
    END_CASE	
END_IF
END_ACTION

ACTION A00_initialization_初始化:
R_TRIG[1](CLK:=%MX2005.5 , Q=> );  //泵空闲中
R_TRIG[2](CLK:=%MX2005.5 , Q=> );  //泵空闲中

CASE 初始化step OF
	0:
		润洗展缸STEP:=0;
		清洗STEP:=0;
		上液step:=0;
		放硅胶板step:=0;
		展开step:=0;
		expand_initialization_OK:=FALSE;
		Expand_Group_clean_OK:=FALSE;
		Expand_up_liquid_OK:=FALSE;
		Expand_silica_gel_plate_OK:=FALSE;
		展开工位允许放硅胶板:=FALSE;
		展开工位允许取硅胶板:=FALSE;
		展开工位机器人到达准备点:=FALSE;
		展开工位机器人放硅胶板完成:=FALSE;
		展开工位取硅胶板完成:=FALSE;
		展开工位允许放硅胶板1:=FALSE;
		CASE Expand_Group OF
			1:
				CASE Expand_Number OF
					1:
						展缸1气缸1手动:=FALSE;
						展缸1气缸1自动:=FALSE;
						展缸1进液电池阀1手动:=FALSE;
						展缸1进液电池阀1自动:=FALSE;
						展缸1排液电池阀1手动:=FALSE;
						展缸1排液电池阀1自动:=FALSE;
						展缸1吹气电池阀1手动:=FALSE;
						展缸1吹气电池阀1自动:=FALSE;
					2:
						展缸1气缸2手动:=FALSE;
						展缸1气缸2自动:=FALSE;
						展缸1进液电池阀2手动:=FALSE;
						展缸1进液电池阀2自动:=FALSE;
						展缸1排液电池阀2手动:=FALSE;
						展缸1排液电池阀2自动:=FALSE;
						展缸1吹气电池阀2手动:=FALSE;
						展缸1吹气电池阀2自动:=FALSE;	
					3:
						展缸1气缸3手动:=FALSE;
						展缸1气缸3自动:=FALSE;
						展缸1进液电池阀3手动:=FALSE;
						展缸1进液电池阀3自动:=FALSE;	
						展缸1排液电池阀3手动:=FALSE;
						展缸1排液电池阀3自动:=FALSE;
						展缸1吹气电池阀3手动:=FALSE;
						展缸1吹气电池阀3自动:=FALSE;	
					4:
						展缸1气缸4手动:=FALSE;
						展缸1气缸4自动:=FALSE;
						展缸1进液电池阀4手动:=FALSE;
						展缸1进液电池阀4自动:=FALSE;	
						展缸1排液电池阀4手动:=FALSE;
						展缸1排液电池阀4自动:=FALSE;
						展缸1吹气电池阀4手动:=FALSE;
						展缸1吹气电池阀4自动:=FALSE;	
				END_CASE
				IF %MW1300=0 AND 泵站位符=FALSE  THEN
					转发转存:='/1Z0,2,2R$R';     //泵初始化指令 
					%MW1300:=LEN(STR:= 转发转存);   //发送字节数
					泵站位符:=TRUE;
					初始化STEP:=10;
				END_IF
			2:
				CASE Expand_Number OF
					1:
						展缸2气缸1手动:=FALSE;
						展缸2气缸1自动:=FALSE;
						展缸2进液电池阀1手动:=FALSE;
						展缸2进液电池阀1自动:=FALSE;
						展缸2排液电池阀1手动:=FALSE;
						展缸2排液电池阀1自动:=FALSE;
						展缸2吹气电池阀1手动:=FALSE;
						展缸2吹气电池阀1自动:=FALSE;
					2:
						展缸2气缸2手动:=FALSE;
						展缸2气缸2自动:=FALSE;
						展缸2进液电池阀2手动:=FALSE;
						展缸2进液电池阀2自动:=FALSE;
						展缸2排液电池阀2手动:=FALSE;
						展缸2排液电池阀2自动:=FALSE;
						展缸2吹气电池阀2手动:=FALSE;
						展缸2吹气电池阀2自动:=FALSE;	
					3:
						展缸2气缸3手动:=FALSE;
						展缸2气缸3自动:=FALSE;
						展缸2进液电池阀3手动:=FALSE;
						展缸2进液电池阀3自动:=FALSE;	
						展缸2排液电池阀3手动:=FALSE;
						展缸2排液电池阀3自动:=FALSE;
						展缸2吹气电池阀3手动:=FALSE;
						展缸2吹气电池阀3自动:=FALSE;	
					4:
						展缸2气缸4手动:=FALSE;
						展缸2气缸4自动:=FALSE;
						展缸2进液电池阀4手动:=FALSE;
						展缸2进液电池阀4自动:=FALSE;	
						展缸2排液电池阀4手动:=FALSE;
						展缸2排液电池阀4自动:=FALSE;
						展缸2吹气电池阀4手动:=FALSE;
						展缸2吹气电池阀4自动:=FALSE;
				END_CASE 
				 IF %MW1300=0 AND 泵站位符=FALSE  THEN
					转发转存:='/2Z0,2,2R$R';     //泵初始化指令 
					%MW1300:=LEN(STR:= 转发转存);   //发送字节数
					泵站位符:=TRUE;
					初始化STEP:=10;
				END_IF
		END_CASE

		展开工位允许放硅胶板:=FALSE;
	
		
		
	10:
		CASE Expand_Group OF
			1:
				IF %MW1300=0 THEN
					转发转存:='/1Q$R';          //查询泵状态指令
					%MW1300:=LEN(STR:= 转发转存);
				END_IF
				
				
				IF R_TRIG[1].Q THEN
					泵初始化完成:=TRUE;
					泵站位符:=FALSE;
					初始化STEP:=0;
				END_IF
			2:
				IF %MW1300=0 THEN
					转发转存:='/2Q$R';          //查询泵状态指令
					%MW1300:=LEN(STR:= 转发转存);
				END_IF
				
				IF R_TRIG[2].Q THEN
					泵初始化完成:=TRUE;
					泵站位符:=FALSE;
					初始化STEP:=0;
				END_IF
		END_CASE
END_CASE
END_ACTION

ACTION A10_pipeline_cleaning_清洗管路:
TON[2](IN:=清洗STEP=10,PT:=T#1S);
TON_0(IN:=清洗STEP=20, PT:=T#3S , Q=> , ET=> );
R_TRIG[5](CLK:=%MX2005.5 , Q=> );  //泵空闲中
CASE 清洗STEP OF
	0 :
		大真空泵站位[10]:=TRUE;
		IF %MW1300=0 AND 泵站位符=FALSE  THEN
			转发转存:=Expand_forward_instructions; 
			%MW1300:=LEN(STR:= 转发转存);   //发送字节数
			泵站位符:=TRUE;
			清洗STEP:=10;
		END_IF
	10:
		//TON[2](IN:=TRUE,PT:=T#1S);
		IF %MW1300=0 AND TON[2].Q THEN
			CASE Expand_Group OF
				1:
					转发转存:='/1Q$R';          //查询泵状态指令
				2:
					转发转存:='/2Q$R';          //查询泵状态指令
			END_CASE
			%MW1300:=LEN(STR:= 转发转存);
		END_IF
		
		
		IF R_TRIG[5].Q THEN
			泵站位符:=FALSE;
			清洗STEP:=20;
		END_IF
	20:
		
		IF TON_0.Q THEN
			大真空泵站位[10]:=FALSE;
			转发转存:='';
			%MW1300:=128;
			Expand_Group_clean_OK:=TRUE;
			清洗STEP:=0;
		END_IF

		
END_CASE
END_ACTION

END_PROGRAM

// Device/Application/40_Man/Photo_scraper_拍照刮板
PROGRAM Photo_scraper_拍照刮板
VAR
	初始化step: INT;
	拍照step: INT;
	刮板收集step: INT;
	机器人取物料step: INT;
	TON_0: TON;
	stepTimer           : TON;       // 步骤内通用定时器（调试期模拟，实机替换为FB完成信号）
    confirmLatched      : BOOL;      // Confirm 上升沿检测：上一周期 Confirm 值
    confirmRisingEdge   : BOOL;      // Confirm 上升沿脉冲（单周期有效）
    phaseA_done_15      : BOOL;      // Step 15 送板完成标志（Phase A 门控）
    phaseA_done_20      : BOOL;      // Step 20 送板完成标志（Phase A 门控）
	k_pass: INT;
	g_plate_surface_z: REAL := 20.5;
	g_total_depth: REAL := 1.0;
END_VAR

// ══════════════════════════════════════════════════════════════
// 刮板工位序列器 — v1.6（协议 v1.6，乒乓握手 + G-code 驱动 + PhotoMode 路由）
// ══════════════════════════════════════════════════════════════
// 对应上位机 Stage: scrape（PLC 变量前缀 scrape）
// 子步 {0, 10, 15, 20, 30, 40, 90}
// 职责：执行拍照刮板全流程（初始化→点样后拍照/展开后拍照→刮取→收集）
//
// 协议要点（v1.6 PhotoMode 路由机制）：
//   - scrape_PhotoMode 控制初始化后的路径选择：
//     0 = 完整刮板模式（默认）：Step 10 → Step 20（展开后拍照+视觉+刮取）
//     1 = 仅 before-photo 模式：Step 10 → Step 15（点样后拍照，乒乓等待后结束）
//   - Step 15 为 before-photo 乒乓等待点：PLC 完成送板后停在 Step 15，
//     等待 PC 侧拍照完成 → 写 scrape_Confirm=TRUE → PLC 归位后 Done
//   - Step 20 为完整刮板乒乓等待点（与 v1.5 一致）
//   - PhotoMode 由 PC 写入，Step 10 路由决策完成后消费归零（不在 Step 0 归零）
//
// v1.5→v1.6 变更：
//   + 新增 scrape_PhotoMode (INT) 变量
//   + 新增 Step 15 (before-photo 乒乓等待)
//   + Step 10 初始化后按 PhotoMode 路由
//   + 子步号扩展为 {0, 10, 15, 20, 30, 40, 90}
//
// 参照 plc_spotting.txt（spotting 工位）模板编写
// ══════════════════════════════════════════════════════════════
//
// ★★★ PLC工程师交付清单 ★★★
// ─────────────────────────────────────────────────────────────
// 交付状态：v1.6 正式交付（2026-05-17）
// 协议版本：v1.6（对应文档 docs/PLC_Unified_Stage_Protocol.md §8）
// Mock 联调：已通过上位机 mock plc_server 联调验证
// ─────────────────────────────────────────────────────────────
// 1. 新增 GVL 变量（必须添加到全局变量表）：
//    scrape_PhotoMode : INT  — 拍照模式选择（0=完整刮板, 1=仅before-photo）
//    其余 scrape_* 变量与 v1.5 一致，见 VAR_GLOBAL 声明
//
// 2. 关键实机集成点（搜索 TODO【实机集成点】）：
//    □ Step 10: 初始化 FB 替换（当前 stepTimer PT:=T#5S 模拟）
//    □ Step 15 Phase A: 送板入拍照位 FB（点样后送板→拍照→回转运位）
//    □ Step 15 归位: 送板回转运位（Confirm 后板需回到转运位待展开）
//    □ Step 20 Phase A: 送板入拍照位 FB（展开后送板→拍照→刮取）
//    □ Step 30: G-code 解析器 + 刮板运动 FB
//    □ Step 40: 机器人取粉末收集器 FB
//
// 3. 关键安全判断（搜索 TODO【逻辑判断】）：
//    □ 急停时停止刮板电机 + 关闭相机触发
//    □ 复位时清空运动指令
//    □ Step 30 安全占位 G-code 识别（"G0 Z10.0\nM2\n" → 跳过刮板）
//    □ 各步骤超时保护
//
// 4. Phase A 门控机制说明：
//    Step 15/20 的 Confirm 上升沿检测带 phaseA_done 门控标志，
//    确保 PLC 完成送板动作后才检测 PC 侧 Confirm 信号，
//    防止 PC 提前写 Confirm 导致板未到位就推进。
//
// 6. 验收检查清单（实机集成后逐项确认）：
//    □ scrape_PhotoMode=0：FSM 轨迹 0→10→20→30→40→0+Done
//    □ scrape_PhotoMode=1：FSM 轨迹 0→10→15→0+Done
//    □ Step 15 乒乓：PC 写 Confirm=TRUE 后 FSM 归位+Done
//    □ Step 20 乒乓：PC 写 Confirm=TRUE 后 FSM 推进到 Step 30
//    □ Phase A 门控：Step 15/20 送板完成前 Confirm 不触发推进
//    □ 安全占位 G-code：Step 30 收到 "G0 Z10.0\nM2\n" 时跳过刮板
//    □ 急停联锁：PLC_EStop=TRUE 时所有动作停止 + Error 置位
//    □ Reset 脉冲：scrape_Reset=TRUE→FALSE 后 Step/Error 清零
//    □ Enable=FALSE 清 Done：上位机拉低 Enable 后 Done 自动归零
// ─────────────────────────────────────────────────────────────
//
// ★★★ 调试期说明 ★★★
// 本文件为调试期简化版，所有 stepTimer 模拟的位置均为实机集成点。
// 标记说明：
//   TODO【实机集成点】— 需替换为真实 FB/IO 调用的占位
//   TODO【逻辑判断】  — 实机必须增加的条件检查/安全守卫
//   当前 stepTimer PT:=T#5S 仅为模拟延时，实机应替换为实际完成条件
// ══════════════════════════════════════════════════════════════

// ── 1. 急停联锁（最高优先级）──
// TODO【逻辑判断】实机急停时应额外执行：
//   - 停止当前正在执行的刮板电机（若有运动控制）
//   - 关闭相机触发信号
//   - 若 Step 30 正在执行 G-code 路径，急停运动轴
IF NOT 急停 THEN
    scrape_Step  := 0;
    scrape_Done  := FALSE;
    scrape_Error := TRUE;
    scrape_Busy  := FALSE;
    confirmLatched  := FALSE;
    confirmRisingEdge := FALSE;
    phaseA_done_15  := FALSE;
    phaseA_done_20  := FALSE;
	刮板拍照真空自动:=FALSE;
	刮板拍照无刷电机自动:=FALSE;
    stepTimer(IN := FALSE, PT := T#0S);
    RETURN;
END_IF

// ── 2. 复位脉冲（用于错误恢复 / 强制清状态）──
// TODO【逻辑判断】实机复位时应额外执行：
//   - 清空刮板电机运动指令
//   - 复位相机触发状态
IF scrape_Reset THEN
    scrape_Step  := 0;
    scrape_Done  := FALSE;
    scrape_Error := FALSE;
    scrape_Busy  := FALSE;
    confirmLatched  := FALSE;
    confirmRisingEdge := FALSE;
    phaseA_done_15  := FALSE;
    phaseA_done_20  := FALSE;
	初始化step:=0;
	拍照step:=0;
	刮板收集step:=0;
	机器人取物料step:=0;
	 scrape_IsLast := FALSE;       // ★ 新增
	
    stepTimer(IN := FALSE, PT := T#0S);
    RETURN;
END_IF

// ── 3. Enable=FALSE 时清 Done（次周期复位握手）──
//    上位机收到 Done 后会拉低 scrape_Enable，本段确保下一周期 Done 自动归零，
//    避免 Done 残留导致 Step 0 误判。
IF NOT scrape_Enable THEN
    scrape_Done := FALSE;
END_IF

// ── 4. 派生 scrape_Busy（写者唯一：本 POU 是唯一写者，禁止他处赋值）──
scrape_Busy := (scrape_Step >= 10)
            AND (scrape_Step <= 80)
            AND (NOT scrape_Done);

// ── 5. Confirm 上升沿检测（Phase A 门控）──
//    Step 15 / Step 20 乒乓等待期间有效，其余步骤忽略。
//    上升沿 = 当前值为 TRUE 且上一周期为 FALSE。
//
//    ★ Phase A 门控（v1.6.1 修复）★
//    问题：PC 侧 await_stage_step 检测到 Step=15/20 即认为板已到位，会立即写
//          scrape_Confirm=TRUE。但实际上 Step 15/20 入场时 Phase A（送板）尚未完成，
//          phaseA_done_15/20 仍为 FALSE。若每周期无条件更新 confirmLatched，
//          上升沿会被白白消耗——等 Phase A 完成时 confirmRisingEdge 已永远为 FALSE，
//          导致 PLC 卡死在 Step 15/20。
//    修复：仅在 Phase A 完成后才更新 confirmLatched（即"开门"边沿检测），
//          PC 早写的 Confirm=TRUE 会被挂起，等 Phase A 完成后首次进入门控就识别为上升沿。
//    协议契约：PC 端不改，仍按"看到 Step=15/20 即拍照+Confirm"的简洁时序。
IF scrape_Step=15  THEN
    confirmRisingEdge := scrape_Confirm AND (NOT confirmLatched);
    confirmLatched    := scrape_Confirm;
ELSE
    // Phase A 未完成 → 不更新 confirmLatched，保留 PC 早写的 Confirm=TRUE
    confirmRisingEdge := FALSE;
END_IF






// ── 6. 主状态机（刮板序列器，Step 15/20 乒乓握手 + PhotoMode 路由）──
IF MODE_State=1 THEN	
	CASE scrape_Step OF
		0:  // ═══ 空闲：等待 Enable 上升 ═══
			// ★ PhotoMode 不在此归零：消费型变量应在子步内复位，不可在 Step 0 无条件赋值
			//   （否则 PC 写入 PhotoMode=1 后会被 Step 0 每周期覆盖回 0）
			IF scrape_Enable AND (NOT scrape_Done) THEN
				scrape_Step := 10;
				stepTimer(IN := FALSE, PT := T#0S);  // 复位定时器
			END_IF
		10:
			IF scrape_PhotoMode=2 THEN
				scrape_Step := 15;
			ELSE
				A00_initialization_初始化();
				IF Camera_scraper_initialization_OK THEN
					Camera_scraper_initialization_OK:=FALSE;
					scrape_Step := 15;
					拍照工位允许取硅胶板去展开 := FALSE;
				END_IF
			END_IF
				
						
			
		 15: // ═══ before-photo（PhotoMode=1 时经此路径 — 点样后拍照乒乓等待）═══
			// ★ before-photo 乒乓协议 ★
			// PLC 侧：
			//   1. 将硅胶板送至拍照位（送板动作，与 Step 20 Phase A 同理）
			//   2. 送板完成后停在 Step 15，等待 PC 侧 Confirm
			// PC 侧（BeforePhotoStage）：
			//   1. await_stage_step("scrape", 15) — 检测到 Step=15（板已到位信号）
			//   2. 触发相机拍照（保存为 before.jpg，由 CameraService 负责）
			//   3. 写 scrape_Confirm=TRUE → PLC 完成归位
			//
			// 与 Step 20 的区别：
			//   - Step 15 不需要视觉分析 / G-code 下发，仅拍照
			//   - Confirm 后直接归位+Done，不进入刮取流程
			//   - 拍照触发权同 v1.5.1：由上位机 CameraService 负责，PLC 仅执行送板
	
			// ── Phase A：送板执行 ──
			// TODO【实机集成点】替换 stepTimer 为真实 FB 调用：
			//   Material_camera_送板入拍照位 := TRUE;    // 送板动作
			//   等待 Material_camera_送板完成_OK = TRUE
			//   注意：拍照触发不再由 PLC 执行，改由上位机 CameraService 触发
			// TODO【逻辑判断】实机需判断：
			//   - 相机拍照超时保护
			//   - 相机通信故障 → Step 90
			A10_Material_camera_拍照硅胶板();
			stepTimer(IN := FALSE, PT := T#0S);
			phaseA_done_15 := TRUE;  // 标记送板完成
			IF Photo_preparation_completed_OK THEN
				IF scrape_PhotoMode = 1 THEN    ///只拍照
					scrape_Step := 16;  // before-photo 模式：去 Step 15 拍照
					拍照工位允许取硅胶板去展开:=TRUE;
					刮板拍照定位气缸自动:=FALSE;
				ELSIF scrape_PhotoMode=2 OR scrape_PhotoMode=0 THEN
					scrape_Step := 20;  // 完整刮板模式：去 Step 20 拍照+视觉+刮取
					Photo_preparation_completed_OK:=FALSE;
				END_IF
				
				scrape_PhotoMode := 0;  // 消费后复位：路由决策完成后清除 PhotoMode/拍照+刮取
			END_IF
		16:
			IF 取拍照硅胶板完成 THEN
				Photo_preparation_completed_OK:=FALSE;
				取拍照硅胶板完成:=FALSE;
				scrape_Done := TRUE;
				scrape_Step := 0;
			END_IF
	
				// ── Phase B：乒乓等待 — 仅送板完成后检测 Confirm 上升沿 ──
				// PC 侧拍照完成 → 写 Confirm=TRUE → PLC 归位并结束
// 				IF phaseA_done_15 AND confirmRisingEdge THEN
// 					// PC 侧确认：拍照完成
// 					// 消费 Confirm 信号 + 复位 PhotoMode
// 					scrape_Confirm := FALSE;  // PLC 侧消费 Confirm 信号
// 					confirmLatched := FALSE;  // 复位边沿检测，防止下一周期误触发
// 					phaseA_done_15 := FALSE;  // 复位 Phase A 标志
// 					// TODO【实机集成点】归位动作：将板从拍照位送回转运位（待展开）
// 					//   Material_camera_送板回转运位 := TRUE;
// 					//   等待 Material_camera_回位完成_OK = TRUE
// 					// 当前调试期直接归位完成
// 					scrape_Done := TRUE;
// 					scrape_Busy := FALSE;
// 					scrape_Step := 0;
// 				END_IF
			
						

		20: // ═══ 刮取（消费 scrape_gcode_instructions，按 G-code 路径刮板）═══
			// 对应 ref_plc_scraping.txt Step 20: Scraper_collection_刮板收集()
			// 区别：旧版为固定路径刮取，新版由 G-code 驱动灵活路径
			//
			// ★ 视觉失败继续场景 ★
			// 当 PC 侧视觉分析失败但用户选择继续时，PC 会下发安全占位 G-code：
			//   "G0 Z10.0\nM2\n"（Z轴抬至安全位 + 程序结束）
			// PLC 工程师应在 Step 30 中识别此占位指令：
			//   - 方案 A：G-code 解析器遇到 M2 时直接跳过刮板动作，推进到 Step 40
			//   - 方案 B：检查 scrape_gcode_instructions 是否以 "G0 Z" 开头，
			//             若为占位指令则跳过刮板（不驱动电机），仅延时后推进
			// 此场景下流程应正常走到 Step 40（机器人取粉末）+ Done=TRUE，
			// 不执行实际刮板动作，但保证 FSM 完整走完。
			//
			// TODO【实机集成点】替换 stepTimer 为真实 FB 调用：
			//   1. 解析 scrape_gcode_instructions 中的 G-code 指令
			//   2. 按指令序列驱动刮板电机执行运动路径
			//      方案 A：CNC 插补器 FB 逐行消费 G-code
			//      方案 B：上位机预生成运动参数，PLC 直接消费坐标序列
			//   3. 等待运动完成信号（CNC_Done / 刮板到位传感器）
			// TODO【逻辑判断】实机需判断：
			//   - G-code 解析错误 → Step 90 故障
			//   - 刮板运动超时保护
			//   - 刮板电机过载/堵转检测 → Step 90
			IF g_pass_count = 0 THEN
					scrape_Step := 40;
			ELSE
				
				A20_Scraper_collection_刮板收集();
				IF Scraper_collection_completed THEN
					刮板拍照工位站位符:=TRUE;
					scrape_gcode_instructions := '';  // 消费 G-code 指令
					Scraper_collection_completed:=FALSE;
					stepTimer(IN := FALSE, PT := T#0S);
					scrape_Step := 30;
				END_IF
			END_IF
		
		 30: // ═══ 机器人取粉末收集器 ═══
        // 对应 ref_plc_scraping.txt Step 30: Robot_material_retrieval_机器人取粉末收集器()
        // TODO【实机集成点】替换 stepTimer 为真实 FB 调用：
        //   Robot_material_retrieval_机器人取粉末收集器();
        //   等待 Robot_completes_material_retrieval = TRUE
        // TODO【逻辑判断】实机需判断：
        //   - 机器人到位传感器确认
        //   - 机器人抓取超时保护
        //   - 粉末收集器就位检测
			A30_Robot_material_retrieval_机器人取粉末收集器();
			IF Robot_completes_material_retrieval THEN
				stepTimer(IN := FALSE, PT := T#0S);
				scrape_IsLast := FALSE;   // ★ 新增：消费型变量子步内归零
				scrape_Done := TRUE;
				scrape_Busy := FALSE;
				Robot_completes_material_retrieval:=FALSE;
				scrape_Step := 0;
			END_IF

		90: // ═══ 故障态：等待外部 scrape_Reset 脉冲 ═══
			scrape_Error := TRUE;   // 故障态本身不动作，仅等待顶部复位逻辑
					
    END_CASE
END_IF

ACTION A30_Robot_material_retrieval_机器人取粉末收集器:




CASE 机器人取物料step OF
	0:
		拍照工位允许取收集器:=TRUE;
		IF 拍照工位机器人到达收集器夹持位 THEN
			拍照工位允许取收集器:=FALSE;
			刮板拍照下压气缸自动:=FALSE;
			机器人取物料step:=10;
		END_IF
	10:
		IF 刮板拍照下压气缸上位 THEN
			拍照工位机器人退出:=TRUE;
			机器人取物料step:=20;
		END_IF
	20:
		IF 拍照工位机器人退出完成 THEN
			拍照工位机器人退出:=FALSE;
			刮板拍照旋转气缸自动:=FALSE;
			拍照工位机器人退出完成:=FALSE;
			机器人取物料step:=30;
			IF scrape_IsLast THEN
				
				机器人取物料step:=30;                    // ★ 最后一次：去 step 30 清板
			ELSE
				Robot_completes_material_retrieval:=TRUE; // ★ 中间：直接 Done，不清板
				机器人取物料step:=0;
			END_IF
		END_IF
	30:
		IF 拍照工位机器人取硅胶板完成 THEN
			拍照工位允许取硅胶板放废料区:=FALSE;
			拍照工位机器人取硅胶板完成:=FALSE;
			Robot_completes_material_retrieval:=TRUE;
			机器人取物料step:=0;
		END_IF	
END_CASE
END_ACTION

ACTION A10_Material_camera_拍照硅胶板:



CASE 拍照step OF
	0:
		刮板轴9XDATE.fAbsTarget:=335;
		刮板轴9XDATE.xMoveAbs:=TRUE;
		IF 刮板轴9XDATE.bAbMoveDone THEN
			刮板轴9XDATE.xMoveAbs:=FALSE;
			IF scrape_PhotoMode=2 THEN
				scrape_WaitConfirm := TRUE;  // 标记送板完成
				拍照step:=10;
			ELSE
				拍照step:=1;
			END_IF
		END_IF
	
	1:
		拍照工位允许放硅胶板:=TRUE;
		IF 拍照工位放硅胶板完成 THEN
			拍照工位允许放硅胶板:=FALSE;
			拍照工位放硅胶板完成:=FALSE;
			刮板拍照定位气缸自动:=TRUE;
			IF scrape_PhotoMode=1 THEN
				拍照step:=30;
			ELSE 
				拍照step:=10;
			END_IF
			
		END_IF
	10:
		拍照工位允许放收集器:=TRUE;
		IF 拍照工位机器人到达夹持位 THEN
			拍照工位允许放收集器:=FALSE;
			刮板拍照下压气缸自动:=TRUE;
			拍照step:=20;
		END_IF
	20:
		TON_0(IN:=TRUE, PT:=T#1S , Q=> , ET=> );
		IF TON_0.Q THEN
			拍照工位机器人退出工位:=TRUE;
			IF 拍照工位机器人退出工位完成 THEN
				拍照工位机器人退出工位完成:=FALSE;
				拍照工位机器人退出工位:=FALSE;
				刮板拍照下压气缸自动:=TRUE;
				IF scrape_PhotoMode=2 THEN
					scrape_WaitConfirm := FALSE;
					Photo_preparation_completed_OK:=TRUE;
					拍照step:=0;
				ELSE
					拍照step:=30;
				END_IF
				
			END_IF
		END_IF
	30:
		IF 刮板拍照遮光气缸上位  THEN
			拍照轴8YDATE.fAbsTarget:=420;
			拍照轴8YDATE.xMoveAbs:=TRUE;
			IF 拍照轴8YDATE.bAbMoveDone THEN
				拍照轴8YDATE.xMoveAbs:=FALSE;
				刮板拍照遮光气缸自动:=TRUE;
				拍照step:=40;
			END_IF
		END_IF
		
	40:
		IF 刮板拍照遮光气缸下位 THEN
			scrape_WaitConfirm := TRUE;  // 标记送板完成
			
			拍照step:=50;
		END_IF
	50:
		IF confirmRisingEdge THEN
			刮板拍照遮光气缸自动:=FALSE;
			scrape_WaitConfirm := FALSE;
			拍照step:=60;
		END_IF
	60:
		IF 刮板拍照遮光气缸上位 THEN
			拍照轴8YDATE.fAbsTarget:=0;
			拍照轴8YDATE.xMoveAbs:=TRUE;
			IF 拍照轴8YDATE.bAbMoveDone THEN
				拍照轴8YDATE.xMoveAbs:=FALSE;
				Photo_preparation_completed_OK:=TRUE;
				拍照step:=0;
			END_IF
		END_IF
	
	
	
	
	
	
	
	
END_CASE
END_ACTION

ACTION A20_Scraper_collection_刮板收集:


CASE 刮板收集step OF
	0:
		刮板拍照真空自动:=TRUE;
		//刮板拍照无刷电机自动:=TRUE;
		
		// 首次进入：初始化 k 与首 pass 的 Z
		IF k_pass = 0 THEN
			
			k_pass := 1;
			g_pass_z := g_plate_surface_z + g_total_depth / INT_TO_LREAL(g_pass_count);
		END_IF
   
		// 触发 CNC：bExe 直接拉高，PLC 侧已有的 SMC pipeline 自动执行
		 CNC启动:= TRUE;
		刮板收集step:=10;
		// 单 pass 完成 → 推进或退出
		
	10:
		IF CNC完成 THEN
			IF k_pass >= g_pass_count THEN
				CNC启动 := FALSE;
				k_pass := 0;
				刮板收集step:=20;
			ELSE
				k_pass := k_pass + 1;
				g_pass_z := g_plate_surface_z
						  + INT_TO_LREAL(k_pass) * g_total_depth
						  / INT_TO_LREAL(g_pass_count);
				 //Z轴高度计算   安全高度+刮取次数*总需要刮取的高速/需要刮取的次数
				CNC启动 := FALSE;   // 下个扫描周期上面 bExe := TRUE 形成上升沿，pipeline 重跑
				刮板收集step:=0;
			END_IF
		END_IF

	20:
		  IF scrape_IsLast THEN
				拍照工位允许取硅胶板放废料区:=TRUE;   // ★ 仅最后一次刮取后才允许送废料
				scrape_IsLast:=FALSE;
				scrape_PhotoMode:=0;
		  END_IF
		刮板拍照定位气缸自动:=FALSE;
		刮板拍照真空自动:=FALSE;
		刮板拍照无刷电机自动:=FALSE;
		CNC启动:=FALSE;
		刮板拍照旋转气缸自动:=TRUE;
		Scraper_collection_completed:=TRUE;
		刮板收集step:=0;
// 	30:
// 		IF 拍照工位机器人取硅胶板完成 THEN
// 			拍照工位允许取硅胶板:=FALSE;
// 			Scraper_collection_completed:=TRUE;
// 			刮板收集step:=0;
// 		END_IF
	
	
	
	
	
	
	
	
END_CASE
END_ACTION

ACTION A00_initialization_初始化:





CASE 初始化step OF
	0:
		刮板拍照真空自动:=FALSE;
		刮板拍照真空手动:=FALSE;
		刮板拍照无刷电机手动:=FALSE;
		刮板拍照无刷电机自动:=FALSE;
		刮板拍照定位气缸手动:=FALSE;
		刮板拍照定位气缸自动:=FALSE;
		粉末收集器定位手动:=FALSE;
		粉末收集器定位自动:=FALSE;
		刮板拍照遮光气缸手动:=FALSE;
		刮板拍照遮光气缸自动:=FALSE;
		刮板拍照旋转气缸手动:=FALSE;
		刮板拍照旋转气缸自动:=FALSE;
		刮板拍照下压气缸手动:=FALSE;
		刮板拍照下压气缸自动:=FALSE;
		拍照工位允许放硅胶板:=FALSE;
		拍照工位允许放收集器:=FALSE;
		拍照工位机器人退出工位:=FALSE;
		拍照工位允许取收集器:=FALSE;
		拍照工位机器人退出:=FALSE;
		scrape_WaitConfirm := FALSE;
		 scrape_IsLast := FALSE;       // ★ 新增
		拍照工位放硅胶板完成 := FALSE;
		
		拍照工位机器人到达夹持位 := FALSE;
		
		拍照工位机器人退出工位完成 := FALSE;
	
		拍照工位机器人到达收集器夹持位 := FALSE;
		
		拍照工位机器人退出完成 := FALSE;
		拍照工位允许取硅胶板放废料区 := FALSE;
		拍照工位允许取硅胶板去展开 := FALSE;
		拍照工位机器人取硅胶板完成 := FALSE;
		拍照step:=0;
		机器人取物料step:=0;
		刮板收集step:=0;
		
		Camera_scraper_initialization_OK:=FALSE;
		Photo_preparation_completed_OK:=FALSE;
		Scraper_collection_completed:=FALSE;
		Robot_completes_material_retrieval:=FALSE;
		初始化step:=5;
	5:
		刮板轴10ZDATE.xMoveAbs:=FALSE;
		刮板轴9XDATE.xMoveAbs:=FALSE;
		拍照轴8YDATE.xMoveAbs:=FALSE;
		初始化step:=6;
	6:
		刮板轴10ZDATE.fAbsTarget:=0;
		刮板轴10ZDATE.xMoveAbs:=TRUE;
		IF 刮板轴10ZDATE.bAbMoveDone THEN
			刮板轴10ZDATE.xMoveAbs:=FALSE;
			初始化step:=10;
		END_IF
	10:
		刮板轴9XDATE.fAbsTarget:=335;
		刮板轴9XDATE.xMoveAbs:=TRUE;
		IF 刮板轴9XDATE.bAbMoveDone THEN
			刮板轴9XDATE.xMoveAbs:=FALSE;
			初始化step:=20;
		END_IF
	20:
		IF 刮板拍照遮光气缸上位 THEN
			拍照轴8YDATE.fAbsTarget:=0;
			拍照轴8YDATE.xMoveAbs:=TRUE;
			IF 拍照轴8YDATE.bAbMoveDone THEN
				拍照轴8YDATE.xMoveAbs:=FALSE;
				Camera_scraper_initialization_OK:=TRUE;
				初始化step:=0;
			END_IF	
		END_IF		
	
END_CASE
END_ACTION

END_PROGRAM

// Device/Application/40_Man/Robotic_Process_机器人流程
PROGRAM Robotic_Process_机器人流程
VAR
	RB_Control_0: FB_RB_Control;
	
	TON: TON;
	R_TRIG: ARRAY[1..2] OF R_TRIG;
END_VAR


R_TRIG[1](CLK:=collect_Old_Plate_Slot>0);
R_TRIG[2](CLK:=scrape_Old_Plate_Slot>0);
//机器人流程
IF MODE_State=1 THEN	
	IF R_TRIG[1].Q THEN
		收集瓶组站位符:=TRUE;
	END_IF
	IF R_TRIG[2].Q THEN
		收集器组站位符:=TRUE;
	END_IF

	CASE 机器人流程 OF
		0:
			IF Status=0 THEN
				IF 上样点样允许放硅胶板 THEN
					机器人流程:=10;
				ELSIF  上样点样允许取硅胶板 AND scrape_Step=0 AND NOT 刮板拍照工位站位符 THEN 
					机器人流程:=20;
				ELSIF 拍照工位允许取硅胶板去展开 AND (Expand_Step=0 OR Expand_Step=30) THEN
					机器人流程:=30;
				ELSIF 展开工位允许取硅胶板 AND scrape_Step=0 AND NOT 刮板拍照工位站位符 THEN       //刮板拍照空闲
					机器人流程:=40;
				ELSIF scrape_Fetch_Rack_Plate>0 AND NOT 刮板拍照暂存工位传感器 THEN 
					机器人流程:=70;
				ELSIF collect_Fetch_Rack_Plate>0 AND NOT 收集平台暂存工位传感器 THEN
					机器人流程:=60;
				ELSIF collect_Old_Plate_Slot>0 AND 收集平台暂存工位传感器 AND NOT 收集瓶组站位符  THEN
					机器人流程:=80;
				ELSIF scrape_Old_Plate_Slot>0 AND 刮板拍照暂存工位传感器 AND  NOT 收集器组站位符 THEN
					机器人流程:=90;
				ELSIF 拍照工位允许放收集器 AND 刮板拍照暂存工位传感器 AND scrape_Consume_Slot>0 THEN 
					机器人流程:=100;
				ELSIF 拍照工位允许取收集器 AND collect_Step=0 THEN           //收集工位空闲
					机器人流程:=110;
				ELSIF 收集工位允许放收集瓶 AND 收集平台暂存工位传感器 AND collect_Consume_Slot>0 THEN
					机器人流程:=120;
				ELSIF 收集工位允许取收集器 AND collect_Powder_Return_Slot>0 THEN
					机器人流程:=130;
				ELSIF 收集工位允许机器人取收集瓶放暂存工位 AND collect_Consume_Slot>0 THEN
					机器人流程:=140;
				ELSIF 拍照工位允许取硅胶板放废料区 THEN
					机器人流程:=50;
				END_IF
			END_IF
			

	
//	取升降机硅胶板放点样机构上

		10:                                                  
			ParameterList3:=1;                           //取1号吸盘工具
			A00_取放工具();
			IF 取工具完成 THEN
				取工具完成:=FALSE;
				ParameterList3:=0; 
				机器人流程:=11;
			END_IF
		11:
			A10_取升降机硅胶板();
			IF 取升降硅胶板完成 THEN
				取升降硅胶板完成:=FALSE;
				机器人流程:=12;		
			END_IF
		12:
			A15_放点样硅胶板();
			IF 放点样硅胶板完成 THEN
				FunctionID:=0;
				放点样硅胶板完成:=FALSE;
				机器人流程:=0;
			END_IF
			
				




//取点样硅胶板放拍照机构上
		20:
			ParameterList3:=1;                           //取1号吸盘工具
			A00_取放工具();
			IF 取工具完成 THEN
				取工具完成:=FALSE;
				机器人流程:=21;
			END_IF
		21:
			A20_取点样硅胶板();
			IF 取点样硅胶板完成 THEN
				
				机器人流程:=22;
			END_IF
		22:
			IF 拍照工位允许放硅胶板 THEN
				
				机器人流程:=23;
			END_IF
		23:
			A35_放拍照硅胶板();
			IF 放拍照硅胶板完成 THEN
				FunctionID:=0;
				放拍照硅胶板完成:=FALSE;
				机器人流程:=0;
			END_IF




//取拍照机构硅胶板放展缸
		30:
			ParameterList3:=1;                           //取1号吸盘工具
			A00_取放工具();
			IF 取工具完成 THEN
				取工具完成:=FALSE;
				机器人流程:=31;
			END_IF
		31:
			A32_取拍照硅胶板();
			IF 取拍照硅胶板完成 THEN
				
				机器人流程:=32;
			END_IF
		32:
			IF 展开工位允许放硅胶板1 THEN
				机器人流程:=33;
			END_IF
		33:
			A25_放展缸硅胶板();
			IF 展开工位机器人放硅胶板完成 THEN
				FunctionID:=0;
				机器人流程:=0;
			END_IF
				
				



//取展缸硅胶板到拍照刮取机构
		40:
			ParameterList3:=1;                           //取1号吸盘工具
			A00_取放工具();
			IF 取工具完成 THEN
				取工具完成:=FALSE;
				机器人流程:=41;
			END_IF
		41:
			A30_取展缸硅胶板();
			IF 取展缸硅胶板完成 THEN
				取展缸硅胶板完成:=FALSE;
				展开工位允许取硅胶板:=FALSE;
				机器人流程:=42;
			END_IF
		42:
			IF 拍照工位允许放硅胶板 THEN
				机器人流程:=43;
			END_IF
		43:
			A35_放拍照硅胶板();
			IF 放拍照硅胶板完成 THEN
				FunctionID:=0;
				放拍照硅胶板完成:=FALSE;
				机器人流程:=0;
			END_IF
			
			





//取拍照刮取硅胶板放到废料区
		50:
			ParameterList3:=1;                           //取1号吸盘工具
			A00_取放工具();
			IF 取工具完成 THEN
				取工具完成:=FALSE;
				机器人流程:=51;
			END_IF
		51:
			A32_取拍照硅胶板();
			IF 取拍照硅胶板完成 THEN
				取拍照硅胶板完成:=FALSE;
				机器人流程:=52;
			END_IF
		52:
			A65_放废料硅胶板();
			IF 取刮板硅胶板放废料区完成 THEN
				拍照工位允许取硅胶板放废料区:=FALSE;
				取刮板硅胶板放废料区完成:=FALSE;
				FunctionID:=0;
				
				机器人流程:=0;
			END_IF







//取收集瓶组到暂存工位
		60:
			ParameterList3:=2;            //取2号大夹持工具
			A00_取放工具();
			IF 取工具完成 THEN
				取工具完成:=FALSE;
				机器人流程:=61;
			END_IF
		61:
			A41_取收集瓶组放暂存工位();
			IF 取收集瓶组放暂存工位完成 THEN
				collect_Fetch_Rack_Plate:=0;
				FunctionID:=0;
				机器人流程:=0;
				取收集瓶组放暂存工位完成:=FALSE;
			END_IF
			
			





//取收集器组到暂存工位
		70:
			ParameterList3:=2;            //取2号大夹持工具
			A00_取放工具();
			IF 取工具完成 THEN
				取工具完成:=FALSE;
				机器人流程:=71;
			END_IF
		71:
			A40_取收集器组放暂存工位();
			IF 取收集器组放暂存工位完成 THEN
				scrape_Fetch_Rack_Plate:=0;
				FunctionID:=0;
				机器人流程:=0;
				取收集器组放暂存工位完成:=FALSE;
			END_IF
		
		
		
		
		
